LIN {X 0,Y 152.545,Z 875.411,A -85,B 0,C 180,E1 7963.211,E2 7963.211} C_VEL
LIN {X 0,Y 145.581,Z 982.767,A -85,B 0,C 180,E1 7954.617,E2 7954.617} C_VEL
LIN {X 0,Y 143.975,Z 1022.889,A -85,B 0,C 180,E1 7951.06,E2 7951.06} C_VEL
LIN {X 0,Y 142.78,Z 1041.292,A -85,B 0,C 180,E1 7948.656,E2 7948.656} C_VEL
LIN {X 0,Y 141.52,Z 1057.681,A -85,B 0,C 180,E1 7945.736,E2 7945.736} C_VEL
LIN {X 0,Y 140.296,Z 1073.463,A -85,B 0,C 180,E1 7942.12,E2 7942.12} C_VEL
LIN {X 0,Y 139.325,Z 1089.114,A -85,B 0,C 180,E1 7937.533,E2 7937.533} C_VEL
LIN {X 0,Y 138.945,Z 1102.914,A -85,B 0,C 180,E1 7932.458,E2 7932.458} C_VEL
LIN {X 0,Y 139.338,Z 1114.971,A -85,B 0,C 180,E1 7926.998,E2 7926.998} C_VEL
LIN {X 0,Y 141.002,Z 1126.172,A -85,B 0,C 180,E1 7920.804,E2 7920.804} C_VEL
LIN {X 0,Y 144.181,Z 1135.172,A -85,B 0,C 180,E1 7914.819,E2 7914.819} C_VEL
LIN {X 0,Y 149.717,Z 1143.18,A -85,B 0,C 180,E1 7908.434,E2 7908.434} C_VEL
LIN {X 0,Y 156.242,Z 1148.409,A -85,B 0,C 180,E1 7903.255,E2 7903.255} C_VEL
LIN {X 0,Y 163.588,Z 1152.185,A -85,B 0,C 180,E1 7898.854,E2 7898.854} C_VEL
LIN {X 0,Y 173.945,Z 1154.929,A -85,B 0,C 180,E1 7894.088,E2 7894.088} C_VEL
LIN {X 0,Y 185.649,Z 1155.901,A -85,B 0,C 180,E1 7889.934,E2 7889.934} C_VEL
LIN {X 0,Y 197.459,Z 1155.135,A -85,B 0,C 180,E1 7886.53,E2 7886.53} C_VEL
LIN {X 0,Y 181.8,Z 1159.577,A -85,B 0,C 180,E1 7882.364,E2 7882.364} C_VEL
LIN {X 0,Y 167.775,Z 1162.466,A -85,B 0,C 180,E1 7877.134,E2 7877.134} C_VEL
LIN {X 0,Y 156.152,Z 1163.814,A -85,B 0,C 180,E1 7870.771,E2 7870.771} C_VEL
LIN {X 0,Y 147.735,Z 1163.571,A -85,B 0,C 180,E1 7863.703,E2 7863.703} C_VEL
LIN {X 0,Y 142.553,Z 1161.973,A -85,B 0,C 180,E1 7855.771,E2 7855.771} C_VEL
LIN {X 0,Y 141.021,Z 1159.791,A -85,B 0,C 180,E1 7849.675,E2 7849.675} C_VEL
LIN {X 0,Y 139.075,Z 1166.656,A -85,B 0,C 180,E1 7844.994,E2 7844.994} C_VEL
LIN {X 0,Y 138.656,Z 1175.79,A -85,B 0,C 180,E1 7837.869,E2 7837.869} C_VEL
LIN {X 0,Y 139.015,Z 1182.334,A -85,B 0,C 180,E1 7831.643,E2 7831.643} C_VEL
LIN {X 0,Y 138.861,Z 1186.047,A -85,B 0,C 180,E1 7827.105,E2 7827.105} C_VEL
LIN {X 0,Y 138.143,Z 1190.598,A -85,B 0,C 180,E1 7819.569,E2 7819.569} C_VEL
LIN {X 0,Y 139.172,Z 1194.136,A -85,B 0,C 180,E1 7811.411,E2 7811.411} C_VEL
LIN {X 0,Y 139.307,Z 1194.975,A -85,B 0,C 180,E1 7808.234,E2 7808.234} C_VEL
LIN {X 0,Y 138.381,Z 1195.914,A -85,B 0,C 180,E1 7799.239,E2 7799.239} C_VEL
LIN {X 0,Y 139.856,Z 1196.329,A -85,B 0,C 180,E1 7796.802,E2 7796.802} C_VEL
LIN {X 0,Y 154.114,Z 1198.205,A -85,B 0,C 180,E1 7786.029,E2 7786.029} C_VEL
LIN {X 0,Y 160.613,Z 1198.418,A -85,B 0,C 180,E1 7782.633,E2 7782.633} C_VEL
LIN {X 0,Y 145.334,Z 1193.936,A -85,B 0,C 180,E1 7773.404,E2 7773.404} C_VEL
LIN {X 0,Y 135.187,Z 1187.729,A -85,B 0,C 180,E1 7762.629,E2 7762.629} C_VEL
LIN {X 0,Y 130.339,Z 1180.191,A -85,B 0,C 180,E1 7751.515,E2 7751.515} C_VEL
LIN {X 0,Y 129.225,Z 1173.64,A -85,B 0,C 180,E1 7743.558,E2 7743.558} C_VEL
LIN {X 0,Y 129.001,Z 1167.014,A -85,B 0,C 180,E1 7736.84,E2 7736.84} C_VEL
LIN {X 0,Y 129.423,Z 1158.193,A -85,B 0,C 180,E1 7729.324,E2 7729.324} C_VEL
LIN {X 0,Y 131.101,Z 1147.526,A -85,B 0,C 180,E1 7721.788,E2 7721.788} C_VEL
LIN {X 0,Y 134.817,Z 1133.432,A -85,B 0,C 180,E1 7713.588,E2 7713.588} C_VEL
LIN {X 0,Y 139.89,Z 1118.577,A -85,B 0,C 180,E1 7706.619,E2 7706.619} C_VEL
LIN {X 0,Y 146.552,Z 1101.226,A -85,B 0,C 180,E1 7700.12,E2 7700.12} C_VEL
LIN {X 0,Y 154.181,Z 1082.006,A -85,B 0,C 180,E1 7694.503,E2 7694.503} C_VEL
LIN {X 0,Y 162.11,Z 1061.669,A -85,B 0,C 180,E1 7689.847,E2 7689.847} C_VEL
LIN {X 0,Y 169.639,Z 1041.208,A -85,B 0,C 180,E1 7686.161,E2 7686.161} C_VEL
LIN {X 0,Y 177.085,Z 1019.188,A -85,B 0,C 180,E1 7683.034,E2 7683.034} C_VEL
LIN {X 0,Y 184.27,Z 995.291,A -85,B 0,C 180,E1 7680.387,E2 7680.387} C_VEL
LIN {X 0,Y 190.704,Z 970.389,A -85,B 0,C 180,E1 7678.271,E2 7678.271} C_VEL
LIN {X 0,Y 196.151,Z 944.496,A -85,B 0,C 180,E1 7676.635,E2 7676.635} C_VEL
LIN {X 0,Y 218.47,Z 820.524,A -85,B 0,C 180,E1 7670.985,E2 7670.985} C_VEL
LIN {X 0,Y 208.205,Z 799.294,A -85,B 0,C 180,E1 7666.295,E2 7666.295} C_VEL
LIN {X 0,Y 199.26,Z 781.915,A -85,B 0,C 180,E1 7661.693,E2 7661.693} C_VEL
LIN {X 0,Y 190.636,Z 766.045,A -85,B 0,C 180,E1 7656.63,E2 7656.63} C_VEL
LIN {X 0,Y 183.761,Z 754.052,A -85,B 0,C 180,E1 7652.031,E2 7652.031} C_VEL
LIN {X 0,Y 176.635,Z 742.307,A -85,B 0,C 180,E1 7646.516,E2 7646.516} C_VEL
LIN {X 0,Y 170.396,Z 732.497,A -85,B 0,C 180,E1 7640.701,E2 7640.701} C_VEL
LIN {X 0,Y 167.6,Z 728.346,A -85,B 0,C 180,E1 7637.728,E2 7637.728} C_VEL
LIN {X 0,Y 162.392,Z 733.212,A -85,B 0,C 180,E1 7634.397,E2 7634.397} C_VEL
LIN {X 0,Y 159.719,Z 736.002,A -85,B 0,C 180,E1 7632.518,E2 7632.518} C_VEL
LIN {X 0,Y 158.824,Z 736.981,A -85,B 0,C 180,E1 7631.893,E2 7631.893} C_VEL
LIN {X 0,Y 156.607,Z 739.804,A -85,B 0,C 180,E1 7630.324,E2 7630.324} C_VEL
LIN {X 0,Y 155.514,Z 740.538,A -85,B 0,C 180,E1 7629.198,E2 7629.198} C_VEL
LIN {X 0,Y 160.894,Z 759.966,A -85,B 0,C 180,E1 7624.021,E2 7624.021} C_VEL
LIN {X 0,Y 163.391,Z 771.027,A -85,B 0,C 180,E1 7621.395,E2 7621.395} C_VEL
LIN {X 0,Y 155.237,Z 815.549,A -85,B 0,C 180,E1 7614.124,E2 7614.124} C_VEL
LIN {X 0,Y 149.141,Z 851.757,A -85,B 0,C 180,E1 7607.907,E2 7607.907} C_VEL
LIN {X 0,Y 144.614,Z 876.252,A -85,B 0,C 180,E1 7603.729,E2 7603.729} C_VEL
LIN {X 0,Y 137.618,Z 981.604,A -85,B 0,C 180,E1 7594.762,E2 7594.762} C_VEL
LIN {X 0,Y 135.971,Z 1022.857,A -85,B 0,C 180,E1 7590.869,E2 7590.869} C_VEL
LIN {X 0,Y 134.825,Z 1040.561,A -85,B 0,C 180,E1 7588.477,E2 7588.477} C_VEL
LIN {X 0,Y 133.59,Z 1056.825,A -85,B 0,C 180,E1 7585.48,E2 7585.48} C_VEL
LIN {X 0,Y 132.34,Z 1073.426,A -85,B 0,C 180,E1 7581.486,E2 7581.486} C_VEL
LIN {X 0,Y 131.46,Z 1088.714,A -85,B 0,C 180,E1 7576.79,E2 7576.79} C_VEL
LIN {X 0,Y 131.178,Z 1102.082,A -85,B 0,C 180,E1 7571.663,E2 7571.663} C_VEL
LIN {X 0,Y 131.686,Z 1114.224,A -85,B 0,C 180,E1 7565.979,E2 7565.979} C_VEL
LIN {X 0,Y 133.357,Z 1124.834,A -85,B 0,C 180,E1 7559.991,E2 7559.991} C_VEL
LIN {X 0,Y 137.012,Z 1134.809,A -85,B 0,C 180,E1 7553.286,E2 7553.286} C_VEL
LIN {X 0,Y 142.58,Z 1142.712,A -85,B 0,C 180,E1 7547.023,E2 7547.023} C_VEL
LIN {X 0,Y 149.715,Z 1148.569,A -85,B 0,C 180,E1 7541.488,E2 7541.488} C_VEL
LIN {X 0,Y 158.954,Z 1153.231,A -85,B 0,C 180,E1 7536.252,E2 7536.252} C_VEL
LIN {X 0,Y 170.023,Z 1156.128,A -85,B 0,C 180,E1 7531.545,E2 7531.545} C_VEL
LIN {X 0,Y 182.808,Z 1157.266,A -85,B 0,C 180,E1 7527.377,E2 7527.377} C_VEL
LIN {X 0,Y 185.108,Z 1157.286,A -85,B 0,C 180,E1 7526.647,E2 7526.647} C_VEL
LIN {X 0,Y 169.803,Z 1160.339,A -85,B 0,C 180,E1 7522.089,E2 7522.089} C_VEL
LIN {X 0,Y 155.982,Z 1161.959,A -85,B 0,C 180,E1 7516.177,E2 7516.177} C_VEL
LIN {X 0,Y 145.322,Z 1162.022,A -85,B 0,C 180,E1 7509.265,E2 7509.265} C_VEL
LIN {X 0,Y 137.39,Z 1160.473,A -85,B 0,C 180,E1 7500.62,E2 7500.62} C_VEL
LIN {X 0,Y 133.942,Z 1157.464,A -85,B 0,C 180,E1 7491.91,E2 7491.91} C_VEL
LIN {X 0,Y 133.735,Z 1156.95,A -85,B 0,C 180,E1 7490.567,E2 7490.567} C_VEL
LIN {X 0,Y 131.347,Z 1164.22,A -85,B 0,C 180,E1 7485.446,E2 7485.446} C_VEL
LIN {X 0,Y 130.903,Z 1173.526,A -85,B 0,C 180,E1 7477.897,E2 7477.897} C_VEL
LIN {X 0,Y 131.3,Z 1179.858,A -85,B 0,C 180,E1 7471.74,E2 7471.74} C_VEL
LIN {X 0,Y 131.259,Z 1183.443,A -85,B 0,C 180,E1 7467.374,E2 7467.374} C_VEL
LIN {X 0,Y 130.553,Z 1187.547,A -85,B 0,C 180,E1 7460.739,E2 7460.739} C_VEL
LIN {X 0,Y 131.554,Z 1192.034,A -85,B 0,C 180,E1 7450.888,E2 7450.888} C_VEL
LIN {X 0,Y 138.235,Z 1195.9,A -85,B 0,C 180,E1 7438.608,E2 7438.608} C_VEL
LIN {X 0,Y 139.856,Z 1196.329,A -85,B 0,C 180,E1 7436.802,E2 7436.802} C_VEL
LIN {X 0,Y 141.939,Z 1196.799,A -85,B 0,C 180,E1 7433.764,E2 7433.764} C_VEL
LIN {X 0,Y 146.454,Z 1196.812,A -85,B 0,C 180,E1 7425.511,E2 7425.511} C_VEL
LIN {X 0,Y 149.63,Z 1196.99,A -85,B 0,C 180,E1 7423.251,E2 7423.251} C_VEL
LIN {X 0,Y 150.631,Z 1197.048,A -85,B 0,C 180,E1 7422.626,E2 7422.626} C_VEL
LIN {X 0,Y 135.976,Z 1191.87,A -85,B 0,C 180,E1 7412.977,E2 7412.977} C_VEL
LIN {X 0,Y 126.267,Z 1184.926,A -85,B 0,C 180,E1 7401.372,E2 7401.372} C_VEL
LIN {X 0,Y 122.321,Z 1177.694,A -85,B 0,C 180,E1 7390.847,E2 7390.847} C_VEL
LIN {X 0,Y 121.327,Z 1170.66,A -85,B 0,C 180,E1 7382.372,E2 7382.372} C_VEL
LIN {X 0,Y 121.176,Z 1163.572,A -85,B 0,C 180,E1 7375.277,E2 7375.277} C_VEL
LIN {X 0,Y 121.794,Z 1154.615,A -85,B 0,C 180,E1 7367.686,E2 7367.686} C_VEL
LIN {X 0,Y 124.035,Z 1142.661,A -85,B 0,C 180,E1 7359.236,E2 7359.236} C_VEL
LIN {X 0,Y 127.925,Z 1129.407,A -85,B 0,C 180,E1 7351.536,E2 7351.536} C_VEL
LIN {X 0,Y 133.683,Z 1113.533,A -85,B 0,C 180,E1 7344.169,E2 7344.169} C_VEL
LIN {X 0,Y 140.64,Z 1096.154,A -85,B 0,C 180,E1 7337.803,E2 7337.803} C_VEL
LIN {X 0,Y 148.56,Z 1076.816,A -85,B 0,C 180,E1 7332.252,E2 7332.252} C_VEL
LIN {X 0,Y 156.67,Z 1056.425,A -85,B 0,C 180,E1 7327.699,E2 7327.699} C_VEL
LIN {X 0,Y 164.608,Z 1035.106,A -85,B 0,C 180,E1 7323.981,E2 7323.981} C_VEL
LIN {X 0,Y 172.371,Z 1012.171,A -85,B 0,C 180,E1 7320.865,E2 7320.865} C_VEL
LIN {X 0,Y 179.199,Z 989.294,A -85,B 0,C 180,E1 7318.458,E2 7318.458} C_VEL
LIN {X 0,Y 185.667,Z 963.62,A -85,B 0,C 180,E1 7316.403,E2 7316.403} C_VEL
LIN {X 0,Y 191.114,Z 937.113,A -85,B 0,C 180,E1 7314.846,E2 7314.846} C_VEL
LIN {X 0,Y 212.132,Z 823.264,A -85,B 0,C 180,E1 7309.63,E2 7309.63} C_VEL
LIN {X 0,Y 202.61,Z 803.298,A -85,B 0,C 180,E1 7305.02,E2 7305.02} C_VEL
LIN {X 0,Y 194.23,Z 786.71,A -85,B 0,C 180,E1 7300.452,E2 7300.452} C_VEL
LIN {X 0,Y 186.023,Z 771.345,A -85,B 0,C 180,E1 7295.402,E2 7295.402} C_VEL
LIN {X 0,Y 179.795,Z 760.212,A -85,B 0,C 180,E1 7291.009,E2 7291.009} C_VEL
LIN {X 0,Y 173.113,Z 748.879,A -85,B 0,C 180,E1 7285.532,E2 7285.532} C_VEL
LIN {X 0,Y 167.239,Z 739.438,A -85,B 0,C 180,E1 7279.846,E2 7279.846} C_VEL
LIN {X 0,Y 165.416,Z 737.027,A -85,B 0,C 180,E1 7277.905,E2 7277.905} C_VEL
LIN {X 0,Y 161.748,Z 740.522,A -85,B 0,C 180,E1 7275.639,E2 7275.639} C_VEL
LIN {X 0,Y 158.335,Z 744.095,A -85,B 0,C 180,E1 7273.334,E2 7273.334} C_VEL
LIN {X 0,Y 155.532,Z 747.222,A -85,B 0,C 180,E1 7271.362,E2 7271.362} C_VEL
LIN {X 0,Y 154.661,Z 748.187,A -85,B 0,C 180,E1 7270.689,E2 7270.689} C_VEL
LIN {X 0,Y 152.41,Z 751.457,A -85,B 0,C 180,E1 7269.056,E2 7269.056} C_VEL
LIN {X 0,Y 151.088,Z 752.484,A -85,B 0,C 180,E1 7267.696,E2 7267.696} C_VEL
LIN {X 0,Y 155.914,Z 771.479,A -85,B 0,C 180,E1 7262.714,E2 7262.714} C_VEL
LIN {X 0,Y 155.794,Z 773.532,A -85,B 0,C 180,E1 7262.317,E2 7262.317} C_VEL
LIN {X 0,Y 147.3,Z 818.296,A -85,B 0,C 180,E1 7254.768,E2 7254.768} C_VEL
LIN {X 0,Y 141.451,Z 851.732,A -85,B 0,C 180,E1 7248.821,E2 7248.821} C_VEL
LIN {X 0,Y 136.669,Z 877.206,A -85,B 0,C 180,E1 7244.271,E2 7244.271} C_VEL
LIN {X 0,Y 129.58,Z 982.567,A -85,B 0,C 180,E1 7234.691,E2 7234.691} C_VEL
LIN {X 0,Y 127.954,Z 1023.158,A -85,B 0,C 180,E1 7230.581,E2 7230.581} C_VEL
LIN {X 0,Y 126.826,Z 1040.595,A -85,B 0,C 180,E1 7228.086,E2 7228.086} C_VEL
LIN {X 0,Y 125.565,Z 1057.39,A -85,B 0,C 180,E1 7224.815,E2 7224.815} C_VEL
LIN {X 0,Y 124.407,Z 1073.471,A -85,B 0,C 180,E1 7220.699,E2 7220.699} C_VEL
LIN {X 0,Y 123.634,Z 1088.566,A -85,B 0,C 180,E1 7215.786,E2 7215.786} C_VEL
LIN {X 0,Y 123.468,Z 1101.769,A -85,B 0,C 180,E1 7210.488,E2 7210.488} C_VEL
LIN {X 0,Y 124.25,Z 1114.595,A -85,B 0,C 180,E1 7204.143,E2 7204.143} C_VEL
LIN {X 0,Y 126.348,Z 1125.444,A -85,B 0,C 180,E1 7197.723,E2 7197.723} C_VEL
LIN {X 0,Y 130.727,Z 1135.641,A -85,B 0,C 180,E1 7190.595,E2 7190.595} C_VEL
LIN {X 0,Y 136.868,Z 1143.476,A -85,B 0,C 180,E1 7184.309,E2 7184.309} C_VEL
LIN {X 0,Y 145.074,Z 1149.665,A -85,B 0,C 180,E1 7178.489,E2 7178.489} C_VEL
LIN {X 0,Y 155.333,Z 1154.452,A -85,B 0,C 180,E1 7173.21,E2 7173.21} C_VEL
LIN {X 0,Y 167.2,Z 1157.426,A -85,B 0,C 180,E1 7168.641,E2 7168.641} C_VEL
LIN {X 0,Y 172.939,Z 1158.217,A -85,B 0,C 180,E1 7166.739,E2 7166.739} C_VEL
LIN {X 0,Y 157.28,Z 1160.043,A -85,B 0,C 180,E1 7161.431,E2 7161.431} C_VEL
LIN {X 0,Y 144.409,Z 1160.358,A -85,B 0,C 180,E1 7154.922,E2 7154.922} C_VEL
LIN {X 0,Y 133.323,Z 1158.865,A -85,B 0,C 180,E1 7145.794,E2 7145.794} C_VEL
LIN {X 0,Y 127.765,Z 1155.911,A -85,B 0,C 180,E1 7136.485,E2 7136.485} C_VEL
LIN {X 0,Y 126.566,Z 1153.907,A -85,B 0,C 180,E1 7131.546,E2 7131.546} C_VEL
LIN {X 0,Y 123.81,Z 1160.941,A -85,B 0,C 180,E1 7126.412,E2 7126.412} C_VEL
LIN {X 0,Y 123.155,Z 1171.322,A -85,B 0,C 180,E1 7117.834,E2 7117.834} C_VEL
LIN {X 0,Y 123.626,Z 1177.712,A -85,B 0,C 180,E1 7111.384,E2 7111.384} C_VEL
LIN {X 0,Y 123.613,Z 1181.117,A -85,B 0,C 180,E1 7107.212,E2 7107.212} C_VEL
LIN {X 0,Y 122.888,Z 1185.844,A -85,B 0,C 180,E1 7099.208,E2 7099.208} C_VEL
LIN {X 0,Y 124.776,Z 1190.699,A -85,B 0,C 180,E1 7087.868,E2 7087.868} C_VEL
LIN {X 0,Y 132.666,Z 1194.586,A -85,B 0,C 180,E1 7075.522,E2 7075.522} C_VEL
LIN {X 0,Y 146.701,Z 1196.742,A -85,B 0,C 180,E1 7064.852,E2 7064.852} C_VEL
LIN {X 0,Y 149.63,Z 1196.99,A -85,B 0,C 180,E1 7063.251,E2 7063.251} C_VEL
LIN {X 0,Y 149.771,Z 1196.868,A -85,B 0,C 180,E1 7062.441,E2 7062.441} C_VEL
LIN {X 0,Y 148.075,Z 1196.388,A -85,B 0,C 180,E1 7061.462,E2 7061.462} C_VEL
LIN {X 0,Y 144.076,Z 1195.428,A -85,B 0,C 180,E1 7060.353,E2 7060.353} C_VEL
LIN {X 0,Y 134.991,Z 1193.082,A -85,B 0,C 180,E1 7058.39,E2 7058.39} C_VEL
LIN {X 0,Y 131.931,Z 1192.058,A -85,B 0,C 180,E1 7056.952,E2 7056.952} C_VEL
LIN {X 0,Y 120.505,Z 1185.095,A -85,B 0,C 180,E1 7045.241,E2 7045.241} C_VEL
LIN {X 0,Y 114.994,Z 1177.091,A -85,B 0,C 180,E1 7033.077,E2 7033.077} C_VEL
LIN {X 0,Y 113.65,Z 1170.011,A -85,B 0,C 180,E1 7024.047,E2 7024.047} C_VEL
LIN {X 0,Y 113.353,Z 1163.295,A -85,B 0,C 180,E1 7016.839,E2 7016.839} C_VEL
LIN {X 0,Y 113.765,Z 1154.541,A -85,B 0,C 180,E1 7008.862,E2 7008.862} C_VEL
LIN {X 0,Y 115.856,Z 1142.609,A -85,B 0,C 180,E1 6999.817,E2 6999.817} C_VEL
LIN {X 0,Y 119.724,Z 1129.381,A -85,B 0,C 180,E1 6991.585,E2 6991.585} C_VEL
LIN {X 0,Y 125.476,Z 1113.805,A -85,B 0,C 180,E1 6983.878,E2 6983.878} C_VEL
LIN {X 0,Y 132.489,Z 1096.741,A -85,B 0,C 180,E1 6977.231,E2 6977.231} C_VEL
LIN {X 0,Y 140.602,Z 1077.546,A -85,B 0,C 180,E1 6971.411,E2 6971.411} C_VEL
LIN {X 0,Y 149.251,Z 1056.491,A -85,B 0,C 180,E1 6966.509,E2 6966.509} C_VEL
LIN {X 0,Y 157.734,Z 1034.393,A -85,B 0,C 180,E1 6962.548,E2 6962.548} C_VEL
LIN {X 0,Y 165.401,Z 1012.337,A -85,B 0,C 180,E1 6959.499,E2 6959.499} C_VEL
LIN {X 0,Y 172.718,Z 988.427,A -85,B 0,C 180,E1 6956.953,E2 6956.953} C_VEL
LIN {X 0,Y 179.231,Z 963.253,A -85,B 0,C 180,E1 6954.915,E2 6954.915} C_VEL
LIN {X 0,Y 184.757,Z 937.115,A -85,B 0,C 180,E1 6953.361,E2 6953.361} C_VEL
LIN {X 0,Y 205.928,Z 826.034,A -85,B 0,C 180,E1 6948.209,E2 6948.209} C_VEL
LIN {X 0,Y 196.018,Z 805.096,A -85,B 0,C 180,E1 6943.124,E2 6943.124} C_VEL
LIN {X 0,Y 187.656,Z 788.383,A -85,B 0,C 180,E1 6938.199,E2 6938.199} C_VEL
LIN {X 0,Y 179.817,Z 773.471,A -85,B 0,C 180,E1 6932.913,E2 6932.913} C_VEL
LIN {X 0,Y 173.81,Z 762.774,A -85,B 0,C 180,E1 6928.274,E2 6928.274} C_VEL
LIN {X 0,Y 168.474,Z 753.77,A -85,B 0,C 180,E1 6923.53,E2 6923.53} C_VEL
LIN {X 0,Y 164.045,Z 746.262,A -85,B 0,C 180,E1 6918.865,E2 6918.865} C_VEL
LIN {X 0,Y 163.406,Z 745.624,A -85,B 0,C 180,E1 6918.208,E2 6918.208} C_VEL
LIN {X 0,Y 157.789,Z 751.248,A -85,B 0,C 180,E1 6914.717,E2 6914.717} C_VEL
LIN {X 0,Y 154.217,Z 755.191,A -85,B 0,C 180,E1 6912.264,E2 6912.264} C_VEL
LIN {X 0,Y 151.528,Z 758.646,A -85,B 0,C 180,E1 6910.34,E2 6910.34} C_VEL
LIN {X 0,Y 150.314,Z 760.001,A -85,B 0,C 180,E1 6909.312,E2 6909.312} C_VEL
LIN {X 0,Y 147.907,Z 763.623,A -85,B 0,C 180,E1 6907.563,E2 6907.563} C_VEL
LIN {X 0,Y 146.552,Z 764.968,A -85,B 0,C 180,E1 6906.034,E2 6906.034} C_VEL
LIN {X 0,Y 148.624,Z 774.15,A -85,B 0,C 180,E1 6903.645,E2 6903.645} C_VEL
LIN {X 0,Y 139.904,Z 818.134,A -85,B 0,C 180,E1 6895.984,E2 6895.984} C_VEL
LIN {X 0,Y 133.933,Z 850.931,A -85,B 0,C 180,E1 6889.911,E2 6889.911} C_VEL
LIN {X 0,Y 128.735,Z 877.891,A -85,B 0,C 180,E1 6884.844,E2 6884.844} C_VEL
LIN {X 0,Y 121.611,Z 981.542,A -85,B 0,C 180,E1 6874.745,E2 6874.745} C_VEL
LIN {X 0,Y 119.971,Z 1022.989,A -85,B 0,C 180,E1 6870.273,E2 6870.273} C_VEL
LIN {X 0,Y 118.863,Z 1040.253,A -85,B 0,C 180,E1 6867.683,E2 6867.683} C_VEL
LIN {X 0,Y 117.593,Z 1057.641,A -85,B 0,C 180,E1 6864.076,E2 6864.076} C_VEL
LIN {X 0,Y 116.474,Z 1074.17,A -85,B 0,C 180,E1 6859.549,E2 6859.549} C_VEL
LIN {X 0,Y 115.87,Z 1088.027,A -85,B 0,C 180,E1 6854.762,E2 6854.762} C_VEL
LIN {X 0,Y 115.878,Z 1102.165,A -85,B 0,C 180,E1 6848.728,E2 6848.728} C_VEL
LIN {X 0,Y 116.867,Z 1114.218,A -85,B 0,C 180,E1 6842.441,E2 6842.441} C_VEL
LIN {X 0,Y 119.569,Z 1125.934,A -85,B 0,C 180,E1 6835.193,E2 6835.193} C_VEL
LIN {X 0,Y 124.506,Z 1136.018,A -85,B 0,C 180,E1 6827.938,E2 6827.938} C_VEL
LIN {X 0,Y 132.005,Z 1144.596,A -85,B 0,C 180,E1 6820.982,E2 6820.982} C_VEL
LIN {X 0,Y 141.584,Z 1151.073,A -85,B 0,C 180,E1 6814.921,E2 6814.921} C_VEL
LIN {X 0,Y 152.901,Z 1155.882,A -85,B 0,C 180,E1 6809.757,E2 6809.757} C_VEL
LIN {X 0,Y 160.969,Z 1158.005,A -85,B 0,C 180,E1 6806.78,E2 6806.78} C_VEL
LIN {X 0,Y 145.565,Z 1158.571,A -85,B 0,C 180,E1 6800.796,E2 6800.796} C_VEL
LIN {X 0,Y 130.941,Z 1157.271,A -85,B 0,C 180,E1 6791.54,E2 6791.54} C_VEL
LIN {X 0,Y 122.799,Z 1154.407,A -85,B 0,C 180,E1 6781.948,E2 6781.948} C_VEL
LIN {X 0,Y 119.571,Z 1150.659,A -85,B 0,C 180,E1 6772.745,E2 6772.745} C_VEL
LIN {X 0,Y 116.216,Z 1158.257,A -85,B 0,C 180,E1 6767.002,E2 6767.002} C_VEL
LIN {X 0,Y 115.44,Z 1169.328,A -85,B 0,C 180,E1 6757.458,E2 6757.458} C_VEL
LIN {X 0,Y 116.017,Z 1175.925,A -85,B 0,C 180,E1 6750.487,E2 6750.487} C_VEL
LIN {X 0,Y 115.924,Z 1179.23,A -85,B 0,C 180,E1 6746.037,E2 6746.037} C_VEL
LIN {X 0,Y 115.348,Z 1184.244,A -85,B 0,C 180,E1 6736.968,E2 6736.968} C_VEL
LIN {X 0,Y 118.617,Z 1189.473,A -85,B 0,C 180,E1 6723.995,E2 6723.995} C_VEL
LIN {X 0,Y 127.906,Z 1193.185,A -85,B 0,C 180,E1 6711.854,E2 6711.854} C_VEL
LIN {X 0,Y 140.818,Z 1195.288,A -85,B 0,C 180,E1 6702.671,E2 6702.671} C_VEL
LIN {X 0,Y 131.931,Z 1192.058,A -85,B 0,C 180,E1 6696.952,E2 6696.952} C_VEL
LIN {X 0,Y 127.499,Z 1190.265,A -85,B 0,C 180,E1 6694.249,E2 6694.249} C_VEL
LIN {X 0,Y 114.215,Z 1183.944,A -85,B 0,C 180,E1 6686.961,E2 6686.961} C_VEL
LIN {X 0,Y 111.564,Z 1181.851,A -85,B 0,C 180,E1 6684.039,E2 6684.039} C_VEL
LIN {X 0,Y 107.035,Z 1174.16,A -85,B 0,C 180,E1 6672.419,E2 6672.419} C_VEL
LIN {X 0,Y 105.781,Z 1166.674,A -85,B 0,C 180,E1 6662.721,E2 6662.721} C_VEL
LIN {X 0,Y 105.559,Z 1159.013,A -85,B 0,C 180,E1 6654.577,E2 6654.577} C_VEL
LIN {X 0,Y 106.381,Z 1149.317,A -85,B 0,C 180,E1 6645.867,E2 6645.867} C_VEL
LIN {X 0,Y 109.024,Z 1137.287,A -85,B 0,C 180,E1 6636.787,E2 6636.787} C_VEL
LIN {X 0,Y 113.713,Z 1123.117,A -85,B 0,C 180,E1 6628.171,E2 6628.171} C_VEL
LIN {X 0,Y 120.362,Z 1106.532,A -85,B 0,C 180,E1 6620.248,E2 6620.248} C_VEL
LIN {X 0,Y 128.242,Z 1088.34,A -85,B 0,C 180,E1 6613.537,E2 6613.537} C_VEL
LIN {X 0,Y 136.875,Z 1068.437,A -85,B 0,C 180,E1 6607.928,E2 6607.928} C_VEL
LIN {X 0,Y 145.527,Z 1047.57,A -85,B 0,C 180,E1 6603.422,E2 6603.422} C_VEL
LIN {X 0,Y 153.942,Z 1025.464,A -85,B 0,C 180,E1 6599.769,E2 6599.769} C_VEL
LIN {X 0,Y 161.999,Z 1001.826,A -85,B 0,C 180,E1 6596.785,E2 6596.785} C_VEL
LIN {X 0,Y 169.185,Z 977.425,A -85,B 0,C 180,E1 6594.442,E2 6594.442} C_VEL
LIN {X 0,Y 175.516,Z 951.425,A -85,B 0,C 180,E1 6592.598,E2 6592.598} C_VEL
LIN {X 0,Y 199.679,Z 828.821,A -85,B 0,C 180,E1 6586.722,E2 6586.722} C_VEL
LIN {X 0,Y 190.422,Z 808.771,A -85,B 0,C 180,E1 6581.629,E2 6581.629} C_VEL
LIN {X 0,Y 181.964,Z 791.617,A -85,B 0,C 180,E1 6576.314,E2 6576.314} C_VEL
LIN {X 0,Y 174.769,Z 777.605,A -85,B 0,C 180,E1 6571.07,E2 6571.07} C_VEL
LIN {X 0,Y 168.373,Z 765.961,A -85,B 0,C 180,E1 6565.654,E2 6565.654} C_VEL
LIN {X 0,Y 162.703,Z 756.306,A -85,B 0,C 180,E1 6559.998,E2 6559.998} C_VEL
LIN {X 0,Y 161.468,Z 754.227,A -85,B 0,C 180,E1 6558.576,E2 6558.576} C_VEL
LIN {X 0,Y 157.097,Z 758.635,A -85,B 0,C 180,E1 6555.953,E2 6555.953} C_VEL
LIN {X 0,Y 153.81,Z 762.248,A -85,B 0,C 180,E1 6553.773,E2 6553.773} C_VEL
LIN {X 0,Y 150.588,Z 765.962,A -85,B 0,C 180,E1 6551.531,E2 6551.531} C_VEL
LIN {X 0,Y 147.001,Z 770.844,A -85,B 0,C 180,E1 6548.875,E2 6548.875} C_VEL
LIN {X 0,Y 145.762,Z 772.27,A -85,B 0,C 180,E1 6547.804,E2 6547.804} C_VEL
LIN {X 0,Y 143.37,Z 776.355,A -85,B 0,C 180,E1 6545.986,E2 6545.986} C_VEL
LIN {X 0,Y 142.023,Z 779.335,A -85,B 0,C 180,E1 6545.118,E2 6545.118} C_VEL
LIN {X 0,Y 139.02,Z 786.157,A -85,B 0,C 180,E1 6543.063,E2 6543.063} C_VEL
LIN {X 0,Y 130.105,Z 830.483,A -85,B 0,C 180,E1 6534.914,E2 6534.914} C_VEL
LIN {X 0,Y 126.204,Z 851.091,A -85,B 0,C 180,E1 6530.918,E2 6530.918} C_VEL
LIN {X 0,Y 120.796,Z 878.663,A -85,B 0,C 180,E1 6525.456,E2 6525.456} C_VEL
LIN {X 0,Y 113.618,Z 981.222,A -85,B 0,C 180,E1 6514.71,E2 6514.71} C_VEL
LIN {X 0,Y 112.017,Z 1022.578,A -85,B 0,C 180,E1 6509.885,E2 6509.885} C_VEL
LIN {X 0,Y 110.892,Z 1040.325,A -85,B 0,C 180,E1 6507.074,E2 6507.074} C_VEL
LIN {X 0,Y 109.62,Z 1058.308,A -85,B 0,C 180,E1 6503.08,E2 6503.08} C_VEL
LIN {X 0,Y 108.617,Z 1074.672,A -85,B 0,C 180,E1 6498.227,E2 6498.227} C_VEL
LIN {X 0,Y 108.152,Z 1089.225,A -85,B 0,C 180,E1 6492.808,E2 6492.808} C_VEL
LIN {X 0,Y 108.468,Z 1103.18,A -85,B 0,C 180,E1 6486.339,E2 6486.339} C_VEL
LIN {X 0,Y 109.934,Z 1115.448,A -85,B 0,C 180,E1 6479.468,E2 6479.468} C_VEL
LIN {X 0,Y 113.644,Z 1127.737,A -85,B 0,C 180,E1 6471.387,E2 6471.387} C_VEL
LIN {X 0,Y 120.044,Z 1138.176,A -85,B 0,C 180,E1 6463.538,E2 6463.538} C_VEL
LIN {X 0,Y 128.779,Z 1146.491,A -85,B 0,C 180,E1 6456.663,E2 6456.663} C_VEL
LIN {X 0,Y 138.824,Z 1152.478,A -85,B 0,C 180,E1 6451.137,E2 6451.137} C_VEL
LIN {X 0,Y 149.361,Z 1156.728,A -85,B 0,C 180,E1 6446.793,E2 6446.793} C_VEL
LIN {X 0,Y 133.713,Z 1156.014,A -85,B 0,C 180,E1 6439.697,E2 6439.697} C_VEL
LIN {X 0,Y 121.973,Z 1153.849,A -85,B 0,C 180,E1 6430.972,E2 6430.972} C_VEL
LIN {X 0,Y 114.814,Z 1150.184,A -85,B 0,C 180,E1 6420.91,E2 6420.91} C_VEL
LIN {X 0,Y 112.702,Z 1147.284,A -85,B 0,C 180,E1 6414.078,E2 6414.078} C_VEL
LIN {X 0,Y 108.882,Z 1154.803,A -85,B 0,C 180,E1 6408.186,E2 6408.186} C_VEL
LIN {X 0,Y 107.736,Z 1166.174,A -85,B 0,C 180,E1 6397.995,E2 6397.995} C_VEL
LIN {X 0,Y 108.372,Z 1173.118,A -85,B 0,C 180,E1 6390.521,E2 6390.521} C_VEL
LIN {X 0,Y 108.443,Z 1176.273,A -85,B 0,C 180,E1 6386.292,E2 6386.292} C_VEL
LIN {X 0,Y 107.827,Z 1181.02,A -85,B 0,C 180,E1 6377.678,E2 6377.678} C_VEL
LIN {X 0,Y 110.243,Z 1186.181,A -85,B 0,C 180,E1 6365.334,E2 6365.334} C_VEL
LIN {X 0,Y 119.911,Z 1190.807,A -85,B 0,C 180,E1 6351.281,E2 6351.281} C_VEL
LIN {X 0,Y 131.134,Z 1193.062,A -85,B 0,C 180,E1 6342.747,E2 6342.747} C_VEL
LIN {X 0,Y 116.603,Z 1186.077,A -85,B 0,C 180,E1 6330.976,E2 6330.976} C_VEL
LIN {X 0,Y 111.564,Z 1181.851,A -85,B 0,C 180,E1 6324.039,E2 6324.039} C_VEL
LIN {X 0,Y 108.776,Z 1179.344,A -85,B 0,C 180,E1 6320.53,E2 6320.53} C_VEL
LIN {X 0,Y 101.748,Z 1173.204,A -85,B 0,C 180,E1 6313.671,E2 6313.671} C_VEL
LIN {X 0,Y 98.734,Z 1168.898,A -85,B 0,C 180,E1 6308.707,E2 6308.707} C_VEL
LIN {X 0,Y 98.479,Z 1168.004,A -85,B 0,C 180,E1 6307.516,E2 6307.516} C_VEL
LIN {X 0,Y 97.836,Z 1160.903,A -85,B 0,C 180,E1 6298.841,E2 6298.841} C_VEL
LIN {X 0,Y 98.067,Z 1151.639,A -85,B 0,C 180,E1 6289.438,E2 6289.438} C_VEL
LIN {X 0,Y 99.893,Z 1140.77,A -85,B 0,C 180,E1 6280.117,E2 6280.117} C_VEL
LIN {X 0,Y 104.262,Z 1126.396,A -85,B 0,C 180,E1 6270.101,E2 6270.101} C_VEL
LIN {X 0,Y 110.599,Z 1110.476,A -85,B 0,C 180,E1 6261.421,E2 6261.421} C_VEL
LIN {X 0,Y 118.345,Z 1093.012,A -85,B 0,C 180,E1 6254.114,E2 6254.114} C_VEL
LIN {X 0,Y 127.575,Z 1072.554,A -85,B 0,C 180,E1 6247.682,E2 6247.682} C_VEL
LIN {X 0,Y 136.68,Z 1051.5,A -85,B 0,C 180,E1 6242.742,E2 6242.742} C_VEL
LIN {X 0,Y 145.523,Z 1029.38,A -85,B 0,C 180,E1 6238.809,E2 6238.809} C_VEL
LIN {X 0,Y 153.704,Z 1006.639,A -85,B 0,C 180,E1 6235.733,E2 6235.733} C_VEL
LIN {X 0,Y 161.299,Z 982.271,A -85,B 0,C 180,E1 6233.242,E2 6233.242} C_VEL
LIN {X 0,Y 167.858,Z 957.178,A -85,B 0,C 180,E1 6231.318,E2 6231.318} C_VEL
LIN {X 0,Y 175.818,Z 919.286,A -85,B 0,C 180,E1 6229.219,E2 6229.219} C_VEL
LIN {X 0,Y 193.548,Z 831.584,A -85,B 0,C 180,E1 6225.165,E2 6225.165} C_VEL
LIN {X 0,Y 184.774,Z 812.323,A -85,B 0,C 180,E1 6220.022,E2 6220.022} C_VEL
LIN {X 0,Y 176.793,Z 795.738,A -85,B 0,C 180,E1 6214.627,E2 6214.627} C_VEL
LIN {X 0,Y 170.22,Z 782.665,A -85,B 0,C 180,E1 6209.5,E2 6209.5} C_VEL
LIN {X 0,Y 164.707,Z 772.306,A -85,B 0,C 180,E1 6204.527,E2 6204.527} C_VEL
LIN {X 0,Y 159.468,Z 762.996,A -85,B 0,C 180,E1 6198.934,E2 6198.934} C_VEL
LIN {X 0,Y 153.537,Z 769.125,A -85,B 0,C 180,E1 6195.344,E2 6195.344} C_VEL
LIN {X 0,Y 149.43,Z 773.913,A -85,B 0,C 180,E1 6192.609,E2 6192.609} C_VEL
LIN {X 0,Y 146.216,Z 778.003,A -85,B 0,C 180,E1 6190.241,E2 6190.241} C_VEL
LIN {X 0,Y 145.087,Z 779.595,A -85,B 0,C 180,E1 6189.429,E2 6189.429} C_VEL
LIN {X 0,Y 142.943,Z 783.128,A -85,B 0,C 180,E1 6187.941,E2 6187.941} C_VEL
LIN {X 0,Y 139.255,Z 791.242,A -85,B 0,C 180,E1 6185.744,E2 6185.744} C_VEL
LIN {X 0,Y 128.983,Z 818.402,A -85,B 0,C 180,E1 6180.514,E2 6180.514} C_VEL
LIN {X 0,Y 122.726,Z 835.555,A -85,B 0,C 180,E1 6176.112,E2 6176.112} C_VEL
LIN {X 0,Y 120.446,Z 841.963,A -85,B 0,C 180,E1 6173.894,E2 6173.894} C_VEL
LIN {X 0,Y 117.7,Z 854.406,A -85,B 0,C 180,E1 6171.385,E2 6171.385} C_VEL
LIN {X 0,Y 112.771,Z 880.165,A -85,B 0,C 180,E1 6166.002,E2 6166.002} C_VEL
LIN {X 0,Y 105.608,Z 981.467,A -85,B 0,C 180,E1 6154.531,E2 6154.531} C_VEL
LIN {X 0,Y 104.056,Z 1022.541,A -85,B 0,C 180,E1 6149.352,E2 6149.352} C_VEL
LIN {X 0,Y 102.922,Z 1040.83,A -85,B 0,C 180,E1 6146.22,E2 6146.22} C_VEL
LIN {X 0,Y 101.723,Z 1058.684,A -85,B 0,C 180,E1 6141.919,E2 6141.919} C_VEL
LIN {X 0,Y 100.87,Z 1074.251,A -85,B 0,C 180,E1 6136.99,E2 6136.99} C_VEL
LIN {X 0,Y 100.581,Z 1089.518,A -85,B 0,C 180,E1 6130.875,E2 6130.875} C_VEL
LIN {X 0,Y 101.202,Z 1103.427,A -85,B 0,C 180,E1 6123.953,E2 6123.953} C_VEL
LIN {X 0,Y 103.164,Z 1115.914,A -85,B 0,C 180,E1 6116.516,E2 6116.516} C_VEL
LIN {X 0,Y 107.559,Z 1127.987,A -85,B 0,C 180,E1 6108.187,E2 6108.187} C_VEL
LIN {X 0,Y 114.335,Z 1137.991,A -85,B 0,C 180,E1 6100.579,E2 6100.579} C_VEL
LIN {X 0,Y 123.955,Z 1146.672,A -85,B 0,C 180,E1 6093.542,E2 6093.542} C_VEL
LIN {X 0,Y 135.266,Z 1153.228,A -85,B 0,C 180,E1 6087.834,E2 6087.834} C_VEL
LIN {X 0,Y 137.921,Z 1154.377,A -85,B 0,C 180,E1 6086.659,E2 6086.659} C_VEL
LIN {X 0,Y 125.063,Z 1153.011,A -85,B 0,C 180,E1 6080.121,E2 6080.121} C_VEL
LIN {X 0,Y 113.621,Z 1149.882,A -85,B 0,C 180,E1 6070.624,E2 6070.624} C_VEL
LIN {X 0,Y 106.98,Z 1145.145,A -85,B 0,C 180,E1 6059.07,E2 6059.07} C_VEL
LIN {X 0,Y 106.117,Z 1143.584,A -85,B 0,C 180,E1 6055.677,E2 6055.677} C_VEL
LIN {X 0,Y 101.944,Z 1150.566,A -85,B 0,C 180,E1 6050.069,E2 6050.069} C_VEL
LIN {X 0,Y 100.08,Z 1159.399,A -85,B 0,C 180,E1 6042.103,E2 6042.103} C_VEL
LIN {X 0,Y 100.444,Z 1168.308,A -85,B 0,C 180,E1 6032.845,E2 6032.845} C_VEL
LIN {X 0,Y 101.015,Z 1172.792,A -85,B 0,C 180,E1 6027.155,E2 6027.155} C_VEL
LIN {X 0,Y 100.418,Z 1177.018,A -85,B 0,C 180,E1 6019.667,E2 6019.667} C_VEL
LIN {X 0,Y 102.189,Z 1182.802,A -85,B 0,C 180,E1 6006.34,E2 6006.34} C_VEL
LIN {X 0,Y 111.551,Z 1187.971,A -85,B 0,C 180,E1 5991.13,E2 5991.13} C_VEL
LIN {X 0,Y 121.504,Z 1190.422,A -85,B 0,C 180,E1 5982.804,E2 5982.804} C_VEL
LIN {X 0,Y 107.082,Z 1182.517,A -85,B 0,C 180,E1 5969.675,E2 5969.675} C_VEL
LIN {X 0,Y 100.399,Z 1174.483,A -85,B 0,C 180,E1 5956.8,E2 5956.8} C_VEL
LIN {X 0,Y 98.479,Z 1168.004,A -85,B 0,C 180,E1 5947.516,E2 5947.516} C_VEL
LIN {X 0,Y 97.374,Z 1165.12,A -85,B 0,C 180,E1 5944.077,E2 5944.077} C_VEL
LIN {X 0,Y 94.299,Z 1160.092,A -85,B 0,C 180,E1 5939.204,E2 5939.204} C_VEL
LIN {X 0,Y 90.446,Z 1152.16,A -85,B 0,C 180,E1 5931.87,E2 5931.87} C_VEL
LIN {X 0,Y 90.285,Z 1149.678,A -85,B 0,C 180,E1 5929.461,E2 5929.461} C_VEL
LIN {X 0,Y 92.515,Z 1137.382,A -85,B 0,C 180,E1 5918.373,E2 5918.373} C_VEL
LIN {X 0,Y 97.081,Z 1123.46,A -85,B 0,C 180,E1 5908.329,E2 5908.329} C_VEL
LIN {X 0,Y 103.511,Z 1108.074,A -85,B 0,C 180,E1 5899.686,E2 5899.686} C_VEL
LIN {X 0,Y 112.028,Z 1089.63,A -85,B 0,C 180,E1 5891.836,E2 5891.836} C_VEL
LIN {X 0,Y 120.832,Z 1070.761,A -85,B 0,C 180,E1 5885.83,E2 5885.83} C_VEL
LIN {X 0,Y 130.312,Z 1049.52,A -85,B 0,C 180,E1 5880.773,E2 5880.773} C_VEL
LIN {X 0,Y 139.408,Z 1027.378,A -85,B 0,C 180,E1 5876.82,E2 5876.82} C_VEL
LIN {X 0,Y 148.012,Z 1003.846,A -85,B 0,C 180,E1 5873.686,E2 5873.686} C_VEL
LIN {X 0,Y 155.98,Z 978.534,A -85,B 0,C 180,E1 5871.164,E2 5871.164} C_VEL
LIN {X 0,Y 162.812,Z 952.353,A -85,B 0,C 180,E1 5869.251,E2 5869.251} C_VEL
LIN {X 0,Y 187.472,Z 834.317,A -85,B 0,C 180,E1 5863.498,E2 5863.498} C_VEL
LIN {X 0,Y 178.995,Z 815.401,A -85,B 0,C 180,E1 5858.194,E2 5858.194} C_VEL
LIN {X 0,Y 171.465,Z 799.321,A -85,B 0,C 180,E1 5852.678,E2 5852.678} C_VEL
LIN {X 0,Y 165.146,Z 786.346,A -85,B 0,C 180,E1 5847.257,E2 5847.257} C_VEL
LIN {X 0,Y 159.395,Z 775.42,A -85,B 0,C 180,E1 5841.528,E2 5841.528} C_VEL
LIN {X 0,Y 157.393,Z 771.829,A -85,B 0,C 180,E1 5839.25,E2 5839.25} C_VEL
LIN {X 0,Y 152.845,Z 776.614,A -85,B 0,C 180,E1 5836.599,E2 5836.599} C_VEL
LIN {X 0,Y 149.16,Z 780.814,A -85,B 0,C 180,E1 5834.232,E2 5834.232} C_VEL
LIN {X 0,Y 145.041,Z 785.915,A -85,B 0,C 180,E1 5831.394,E2 5831.394} C_VEL
LIN {X 0,Y 143.348,Z 788.725,A -85,B 0,C 180,E1 5830.303,E2 5830.303} C_VEL
LIN {X 0,Y 140.003,Z 795.672,A -85,B 0,C 180,E1 5828.514,E2 5828.514} C_VEL
LIN {X 0,Y 129.341,Z 822.682,A -85,B 0,C 180,E1 5823.523,E2 5823.523} C_VEL
LIN {X 0,Y 122.68,Z 839.8,A -85,B 0,C 180,E1 5819.28,E2 5819.28} C_VEL
LIN {X 0,Y 119.976,Z 846.938,A -85,B 0,C 180,E1 5817.028,E2 5817.028} C_VEL
LIN {X 0,Y 108.882,Z 882.399,A -85,B 0,C 180,E1 5809.488,E2 5809.488} C_VEL
LIN {X 0,Y 104.661,Z 897.529,A -85,B 0,C 180,E1 5806.639,E2 5806.639} C_VEL
LIN {X 0,Y 102.865,Z 904.327,A -85,B 0,C 180,E1 5804.522,E2 5804.522} C_VEL
LIN {X 0,Y 102.539,Z 905.91,A -85,B 0,C 180,E1 5803.837,E2 5803.837} C_VEL
LIN {X 0,Y 97.466,Z 985.873,A -85,B 0,C 180,E1 5793.699,E2 5793.699} C_VEL
LIN {X 0,Y 96.057,Z 1023.785,A -85,B 0,C 180,E1 5788.445,E2 5788.445} C_VEL
LIN {X 0,Y 94.975,Z 1041.473,A -85,B 0,C 180,E1 5785.144,E2 5785.144} C_VEL
LIN {X 0,Y 93.896,Z 1058.89,A -85,B 0,C 180,E1 5780.559,E2 5780.559} C_VEL
LIN {X 0,Y 93.188,Z 1074.776,A -85,B 0,C 180,E1 5775.089,E2 5775.089} C_VEL
LIN {X 0,Y 93.155,Z 1089.663,A -85,B 0,C 180,E1 5768.629,E2 5768.629} C_VEL
LIN {X 0,Y 94.149,Z 1103.531,A -85,B 0,C 180,E1 5761.204,E2 5761.204} C_VEL
LIN {X 0,Y 96.854,Z 1116.649,A -85,B 0,C 180,E1 5752.871,E2 5752.871} C_VEL
LIN {X 0,Y 101.864,Z 1128.133,A -85,B 0,C 180,E1 5744.619,E2 5744.619} C_VEL
LIN {X 0,Y 109.519,Z 1138.297,A -85,B 0,C 180,E1 5736.873,E2 5736.873} C_VEL
LIN {X 0,Y 119.927,Z 1146.993,A -85,B 0,C 180,E1 5729.972,E2 5729.972} C_VEL
LIN {X 0,Y 126.876,Z 1151.295,A -85,B 0,C 180,E1 5726.457,E2 5726.457} C_VEL
LIN {X 0,Y 112.585,Z 1148.27,A -85,B 0,C 180,E1 5717.477,E2 5717.477} C_VEL
LIN {X 0,Y 103.029,Z 1143.804,A -85,B 0,C 180,E1 5706.289,E2 5706.289} C_VEL
LIN {X 0,Y 99.651,Z 1139.848,A -85,B 0,C 180,E1 5697.478,E2 5697.478} C_VEL
LIN {X 0,Y 94.63,Z 1147.527,A -85,B 0,C 180,E1 5691.045,E2 5691.045} C_VEL
LIN {X 0,Y 92.4,Z 1157.096,A -85,B 0,C 180,E1 5681.856,E2 5681.856} C_VEL
LIN {X 0,Y 92.86,Z 1165.606,A -85,B 0,C 180,E1 5672.46,E2 5672.46} C_VEL
LIN {X 0,Y 93.534,Z 1169.865,A -85,B 0,C 180,E1 5666.928,E2 5666.928} C_VEL
LIN {X 0,Y 93.012,Z 1173.989,A -85,B 0,C 180,E1 5659.462,E2 5659.462} C_VEL
LIN {X 0,Y 95.229,Z 1180.195,A -85,B 0,C 180,E1 5644.493,E2 5644.493} C_VEL
LIN {X 0,Y 104.627,Z 1185.399,A -85,B 0,C 180,E1 5629.46,E2 5629.46} C_VEL
LIN {X 0,Y 111.976,Z 1187.397,A -85,B 0,C 180,E1 5622.865,E2 5622.865} C_VEL
LIN {X 0,Y 98.411,Z 1179.19,A -85,B 0,C 180,E1 5609.203,E2 5609.203} C_VEL
LIN {X 0,Y 92.31,Z 1170.829,A -85,B 0,C 180,E1 5595.725,E2 5595.725} C_VEL
LIN {X 0,Y 90.615,Z 1163.897,A -85,B 0,C 180,E1 5585.713,E2 5585.713} C_VEL
LIN {X 0,Y 90.075,Z 1157.19,A -85,B 0,C 180,E1 5577.469,E2 5577.469} C_VEL
LIN {X 0,Y 90.285,Z 1149.678,A -85,B 0,C 180,E1 5569.461,E2 5569.461} C_VEL
LIN {X 0,Y 89.99,Z 1145.954,A -85,B 0,C 180,E1 5565.985,E2 5565.985} C_VEL
LIN {X 0,Y 87.997,Z 1139.186,A -85,B 0,C 180,E1 5560.417,E2 5560.417} C_VEL
LIN {X 0,Y 86.588,Z 1131.276,A -85,B 0,C 180,E1 5554.223,E2 5554.223} C_VEL
LIN {X 0,Y 87.252,Z 1127.583,A -85,B 0,C 180,E1 5551.448,E2 5551.448} C_VEL
LIN {X 0,Y 93.422,Z 1112.419,A -85,B 0,C 180,E1 5541.393,E2 5541.393} C_VEL
LIN {X 0,Y 101.816,Z 1094.58,A -85,B 0,C 180,E1 5532.582,E2 5532.582} C_VEL
LIN {X 0,Y 110.927,Z 1075.775,A -85,B 0,C 180,E1 5525.802,E2 5525.802} C_VEL
LIN {X 0,Y 120.497,Z 1055.43,A -85,B 0,C 180,E1 5520.368,E2 5520.368} C_VEL
LIN {X 0,Y 130.136,Z 1033.281,A -85,B 0,C 180,E1 5516.003,E2 5516.003} C_VEL
LIN {X 0,Y 139.239,Z 1009.95,A -85,B 0,C 180,E1 5512.595,E2 5512.595} C_VEL
LIN {X 0,Y 147.758,Z 984.803,A -85,B 0,C 180,E1 5509.872,E2 5509.872} C_VEL
LIN {X 0,Y 154.979,Z 959.097,A -85,B 0,C 180,E1 5507.835,E2 5507.835} C_VEL
LIN {X 0,Y 162.779,Z 924.484,A -85,B 0,C 180,E1 5505.874,E2 5505.874} C_VEL
LIN {X 0,Y 181.433,Z 837.069,A -85,B 0,C 180,E1 5501.77,E2 5501.77} C_VEL
LIN {X 0,Y 173.633,Z 819.099,A -85,B 0,C 180,E1 5496.452,E2 5496.452} C_VEL
LIN {X 0,Y 166.171,Z 802.796,A -85,B 0,C 180,E1 5490.565,E2 5490.565} C_VEL
LIN {X 0,Y 160.687,Z 791.278,A -85,B 0,C 180,E1 5485.454,E2 5485.454} C_VEL
LIN {X 0,Y 155.758,Z 781.554,A -85,B 0,C 180,E1 5480.117,E2 5480.117} C_VEL
LIN {X 0,Y 155.185,Z 780.864,A -85,B 0,C 180,E1 5479.508,E2 5479.508} C_VEL
LIN {X 0,Y 148.805,Z 787.882,A -85,B 0,C 180,E1 5475.762,E2 5475.762} C_VEL
LIN {X 0,Y 144.869,Z 792.604,A -85,B 0,C 180,E1 5473.199,E2 5473.199} C_VEL
LIN {X 0,Y 141.549,Z 798.838,A -85,B 0,C 180,E1 5471.438,E2 5471.438} C_VEL
LIN {X 0,Y 130.218,Z 826.436,A -85,B 0,C 180,E1 5466.618,E2 5466.618} C_VEL
LIN {X 0,Y 123.029,Z 843.976,A -85,B 0,C 180,E1 5462.461,E2 5462.461} C_VEL
LIN {X 0,Y 120.077,Z 851.105,A -85,B 0,C 180,E1 5460.336,E2 5460.336} C_VEL
LIN {X 0,Y 108.729,Z 885.232,A -85,B 0,C 180,E1 5453.446,E2 5453.446} C_VEL
LIN {X 0,Y 104.157,Z 900.552,A -85,B 0,C 180,E1 5450.695,E2 5450.695} C_VEL
LIN {X 0,Y 101.816,Z 908.388,A -85,B 0,C 180,E1 5448.362,E2 5448.362} C_VEL
LIN {X 0,Y 101.249,Z 910.401,A -85,B 0,C 180,E1 5447.874,E2 5447.874} C_VEL
LIN {X 0,Y 95.701,Z 931.048,A -85,B 0,C 180,E1 5444.619,E2 5444.619} C_VEL
LIN {X 0,Y 92.363,Z 944.261,A -85,B 0,C 180,E1 5441.309,E2 5441.309} C_VEL
LIN {X 0,Y 91.193,Z 949.718,A -85,B 0,C 180,E1 5439.025,E2 5439.025} C_VEL
LIN {X 0,Y 91.055,Z 950.907,A -85,B 0,C 180,E1 5438.355,E2 5438.355} C_VEL
LIN {X 0,Y 88.422,Z 1018.409,A -85,B 0,C 180,E1 5428.385,E2 5428.385} C_VEL
LIN {X 0,Y 87.415,Z 1036.733,A -85,B 0,C 180,E1 5425.022,E2 5425.022} C_VEL
LIN {X 0,Y 86.367,Z 1054.681,A -85,B 0,C 180,E1 5420.307,E2 5420.307} C_VEL
LIN {X 0,Y 85.729,Z 1070.234,A -85,B 0,C 180,E1 5414.853,E2 5414.853} C_VEL
LIN {X 0,Y 85.744,Z 1085.663,A -85,B 0,C 180,E1 5408.029,E2 5408.029} C_VEL
LIN {X 0,Y 86.747,Z 1099.173,A -85,B 0,C 180,E1 5400.646,E2 5400.646} C_VEL
LIN {X 0,Y 89.308,Z 1112.244,A -85,B 0,C 180,E1 5392.265,E2 5392.265} C_VEL
LIN {X 0,Y 94.837,Z 1125.317,A -85,B 0,C 180,E1 5382.817,E2 5382.817} C_VEL
LIN {X 0,Y 102.868,Z 1136.088,A -85,B 0,C 180,E1 5374.667,E2 5374.667} C_VEL
LIN {X 0,Y 114.42,Z 1145.927,A -85,B 0,C 180,E1 5367.182,E2 5367.182} C_VEL
LIN {X 0,Y 116.24,Z 1147.224,A -85,B 0,C 180,E1 5366.094,E2 5366.094} C_VEL
LIN {X 0,Y 102.811,Z 1143.176,A -85,B 0,C 180,E1 5356.017,E2 5356.017} C_VEL
LIN {X 0,Y 94.639,Z 1137.605,A -85,B 0,C 180,E1 5343.315,E2 5343.315} C_VEL
LIN {X 0,Y 93.438,Z 1135.859,A -85,B 0,C 180,E1 5339.479,E2 5339.479} C_VEL
LIN {X 0,Y 88.12,Z 1142.957,A -85,B 0,C 180,E1 5333.389,E2 5333.389} C_VEL
LIN {X 0,Y 85.036,Z 1151.462,A -85,B 0,C 180,E1 5324.982,E2 5324.982} C_VEL
LIN {X 0,Y 85.202,Z 1162.328,A -85,B 0,C 180,E1 5312.681,E2 5312.681} C_VEL
LIN {X 0,Y 86.102,Z 1167.268,A -85,B 0,C 180,E1 5305.996,E2 5305.996} C_VEL
LIN {X 0,Y 85.685,Z 1171.961,A -85,B 0,C 180,E1 5296.494,E2 5296.494} C_VEL
LIN {X 0,Y 89.876,Z 1178.713,A -85,B 0,C 180,E1 5278.967,E2 5278.967} C_VEL
LIN {X 0,Y 101.568,Z 1183.751,A -85,B 0,C 180,E1 5264.047,E2 5264.047} C_VEL
LIN {X 0,Y 102.644,Z 1184.04,A -85,B 0,C 180,E1 5263.007,E2 5263.007} C_VEL
LIN {X 0,Y 90.178,Z 1175.806,A -85,B 0,C 180,E1 5249.216,E2 5249.216} C_VEL
LIN {X 0,Y 84.135,Z 1166.466,A -85,B 0,C 180,E1 5233.765,E2 5233.765} C_VEL
LIN {X 0,Y 82.802,Z 1159.912,A -85,B 0,C 180,E1 5224.17,E2 5224.17} C_VEL
LIN {X 0,Y 82.318,Z 1152.065,A -85,B 0,C 180,E1 5214.439,E2 5214.439} C_VEL
LIN {X 0,Y 83.387,Z 1141.469,A -85,B 0,C 180,E1 5203.291,E2 5203.291} C_VEL
LIN {X 0,Y 87.252,Z 1127.583,A -85,B 0,C 180,E1 5191.448,E2 5191.448} C_VEL
LIN {X 0,Y 88.16,Z 1122.482,A -85,B 0,C 180,E1 5187.722,E2 5187.722} C_VEL
LIN {X 0,Y 88.344,Z 1107.363,A -85,B 0,C 180,E1 5177.911,E2 5177.911} C_VEL
LIN {X 0,Y 89.957,Z 1102.448,A -85,B 0,C 180,E1 5175.182,E2 5175.182} C_VEL
LIN {X 0,Y 99.074,Z 1084.353,A -85,B 0,C 180,E1 5167.15,E2 5167.15} C_VEL
LIN {X 0,Y 109.237,Z 1063.983,A -85,B 0,C 180,E1 5160.661,E2 5160.661} C_VEL
LIN {X 0,Y 119.296,Z 1042.469,A -85,B 0,C 180,E1 5155.734,E2 5155.734} C_VEL
LIN {X 0,Y 128.805,Z 1020.035,A -85,B 0,C 180,E1 5151.957,E2 5151.957} C_VEL
LIN {X 0,Y 137.502,Z 996.735,A -85,B 0,C 180,E1 5149.064,E2 5149.064} C_VEL
LIN {X 0,Y 145.362,Z 972.069,A -85,B 0,C 180,E1 5146.798,E2 5146.798} C_VEL
LIN {X 0,Y 152.099,Z 946.278,A -85,B 0,C 180,E1 5145.058,E2 5145.058} C_VEL
LIN {X 0,Y 175.592,Z 839.999,A -85,B 0,C 180,E1 5139.982,E2 5139.982} C_VEL
LIN {X 0,Y 168.638,Z 823.644,A -85,B 0,C 180,E1 5134.92,E2 5134.92} C_VEL
LIN {X 0,Y 161.917,Z 808.334,A -85,B 0,C 180,E1 5129.171,E2 5129.171} C_VEL
LIN {X 0,Y 156.626,Z 796.722,A -85,B 0,C 180,E1 5123.837,E2 5123.837} C_VEL
LIN {X 0,Y 153.186,Z 789.897,A -85,B 0,C 180,E1 5119.94,E2 5119.94} C_VEL
LIN {X 0,Y 148.202,Z 795.307,A -85,B 0,C 180,E1 5117.097,E2 5117.097} C_VEL
LIN {X 0,Y 145.15,Z 798.876,A -85,B 0,C 180,E1 5115.206,E2 5115.206} C_VEL
LIN {X 0,Y 142.362,Z 804.299,A -85,B 0,C 180,E1 5113.983,E2 5113.983} C_VEL
LIN {X 0,Y 130.992,Z 831.041,A -85,B 0,C 180,E1 5109.509,E2 5109.509} C_VEL
LIN {X 0,Y 123.526,Z 848.344,A -85,B 0,C 180,E1 5105.567,E2 5105.567} C_VEL
LIN {X 0,Y 120.567,Z 855.233,A -85,B 0,C 180,E1 5103.636,E2 5103.636} C_VEL
LIN {X 0,Y 109.016,Z 888.062,A -85,B 0,C 180,E1 5097.401,E2 5097.401} C_VEL
LIN {X 0,Y 104.002,Z 903.792,A -85,B 0,C 180,E1 5094.723,E2 5094.723} C_VEL
LIN {X 0,Y 100.949,Z 913.349,A -85,B 0,C 180,E1 5092.156,E2 5092.156} C_VEL
LIN {X 0,Y 94.995,Z 934.024,A -85,B 0,C 180,E1 5089.081,E2 5089.081} C_VEL
LIN {X 0,Y 91.247,Z 947.604,A -85,B 0,C 180,E1 5085.792,E2 5085.792} C_VEL
LIN {X 0,Y 89.469,Z 954.098,A -85,B 0,C 180,E1 5083.178,E2 5083.178} C_VEL
LIN {X 0,Y 84.475,Z 971.673,A -85,B 0,C 180,E1 5079.27,E2 5079.27} C_VEL
LIN {X 0,Y 82.379,Z 979.188,A -85,B 0,C 180,E1 5076.475,E2 5076.475} C_VEL
LIN {X 0,Y 81.615,Z 982.675,A -85,B 0,C 180,E1 5074.283,E2 5074.283} C_VEL
LIN {X 0,Y 81.57,Z 983.955,A -85,B 0,C 180,E1 5073.059,E2 5073.059} C_VEL
LIN {X 0,Y 80.376,Z 1022.244,A -85,B 0,C 180,E1 5066.638,E2 5066.638} C_VEL
LIN {X 0,Y 79.467,Z 1039.391,A -85,B 0,C 180,E1 5062.941,E2 5062.941} C_VEL
LIN {X 0,Y 78.614,Z 1056.648,A -85,B 0,C 180,E1 5057.756,E2 5057.756} C_VEL
LIN {X 0,Y 78.259,Z 1073.484,A -85,B 0,C 180,E1 5051.033,E2 5051.033} C_VEL
LIN {X 0,Y 78.822,Z 1088.129,A -85,B 0,C 180,E1 5043.621,E2 5043.621} C_VEL
LIN {X 0,Y 80.693,Z 1102.241,A -85,B 0,C 180,E1 5035.009,E2 5035.009} C_VEL
LIN {X 0,Y 84.737,Z 1115.579,A -85,B 0,C 180,E1 5025.638,E2 5025.638} C_VEL
LIN {X 0,Y 91.92,Z 1128.147,A -85,B 0,C 180,E1 5016.252,E2 5016.252} C_VEL
LIN {X 0,Y 102.185,Z 1139.092,A -85,B 0,C 180,E1 5008.089,E2 5008.089} C_VEL
LIN {X 0,Y 106.135,Z 1142.374,A -85,B 0,C 180,E1 5005.601,E2 5005.601} C_VEL
LIN {X 0,Y 93.792,Z 1137.426,A -85,B 0,C 180,E1 4994.399,E2 4994.399} C_VEL
LIN {X 0,Y 87.367,Z 1131.859,A -85,B 0,C 180,E1 4981.755,E2 4981.755} C_VEL
LIN {X 0,Y 81.036,Z 1139.675,A -85,B 0,C 180,E1 4974.793,E2 4974.793} C_VEL
LIN {X 0,Y 77.428,Z 1148.898,A -85,B 0,C 180,E1 4964.957,E2 4964.957} C_VEL
LIN {X 0,Y 77.576,Z 1158.813,A -85,B 0,C 180,E1 4952.945,E2 4952.945} C_VEL
LIN {X 0,Y 78.761,Z 1164.47,A -85,B 0,C 180,E1 4944.892,E2 4944.892} C_VEL
LIN {X 0,Y 78.511,Z 1169.23,A -85,B 0,C 180,E1 4934.477,E2 4934.477} C_VEL
LIN {X 0,Y 82.69,Z 1175.375,A -85,B 0,C 180,E1 4917.845,E2 4917.845} C_VEL
LIN {X 0,Y 93.472,Z 1180.35,A -85,B 0,C 180,E1 4903.223,E2 4903.223} C_VEL
LIN {X 0,Y 81.295,Z 1171.358,A -85,B 0,C 180,E1 4887.881,E2 4887.881} C_VEL
LIN {X 0,Y 76.172,Z 1162.206,A -85,B 0,C 180,E1 4872.14,E2 4872.14} C_VEL
LIN {X 0,Y 74.977,Z 1155.604,A -85,B 0,C 180,E1 4862.309,E2 4862.309} C_VEL
LIN {X 0,Y 74.72,Z 1146.455,A -85,B 0,C 180,E1 4850.776,E2 4850.776} C_VEL
LIN {X 0,Y 76.652,Z 1134.946,A -85,B 0,C 180,E1 4838.595,E2 4838.595} C_VEL
LIN {X 0,Y 81.65,Z 1120.493,A -85,B 0,C 180,E1 4826.397,E2 4826.397} C_VEL
LIN {X 0,Y 89.196,Z 1104.023,A -85,B 0,C 180,E1 4815.991,E2 4815.991} C_VEL
LIN {X 0,Y 89.957,Z 1102.448,A -85,B 0,C 180,E1 4815.182,E2 4815.182} C_VEL
LIN {X 0,Y 91.841,Z 1096.713,A -85,B 0,C 180,E1 4812.196,E2 4812.196} C_VEL
LIN {X 0,Y 94.302,Z 1080.166,A -85,B 0,C 180,E1 4804.068,E2 4804.068} C_VEL
LIN {X 0,Y 96.423,Z 1074.771,A -85,B 0,C 180,E1 4801.978,E2 4801.978} C_VEL
LIN {X 0,Y 107.135,Z 1053.575,A -85,B 0,C 180,E1 4796.025,E2 4796.025} C_VEL
LIN {X 0,Y 117.237,Z 1031.844,A -85,B 0,C 180,E1 4791.653,E2 4791.653} C_VEL
LIN {X 0,Y 126.855,Z 1008.536,A -85,B 0,C 180,E1 4788.267,E2 4788.267} C_VEL
LIN {X 0,Y 135.509,Z 984.301,A -85,B 0,C 180,E1 4785.689,E2 4785.689} C_VEL
LIN {X 0,Y 142.987,Z 959.249,A -85,B 0,C 180,E1 4783.726,E2 4783.726} C_VEL
LIN {X 0,Y 151.393,Z 923.937,A -85,B 0,C 180,E1 4781.773,E2 4781.773} C_VEL
LIN {X 0,Y 169.774,Z 842.721,A -85,B 0,C 180,E1 4778.024,E2 4778.024} C_VEL
LIN {X 0,Y 163.007,Z 826.408,A -85,B 0,C 180,E1 4772.659,E2 4772.659} C_VEL
LIN {X 0,Y 156.875,Z 811.944,A -85,B 0,C 180,E1 4766.899,E2 4766.899} C_VEL
LIN {X 0,Y 152.193,Z 801.354,A -85,B 0,C 180,E1 4761.695,E2 4761.695} C_VEL
LIN {X 0,Y 151.054,Z 798.94,A -85,B 0,C 180,E1 4760.288,E2 4760.288} C_VEL
LIN {X 0,Y 145.888,Z 804.748,A -85,B 0,C 180,E1 4757.428,E2 4757.428} C_VEL
LIN {X 0,Y 143.862,Z 808.774,A -85,B 0,C 180,E1 4756.624,E2 4756.624} C_VEL
LIN {X 0,Y 131.837,Z 836.18,A -85,B 0,C 180,E1 4752.261,E2 4752.261} C_VEL
LIN {X 0,Y 124.022,Z 853.485,A -85,B 0,C 180,E1 4748.432,E2 4748.432} C_VEL
LIN {X 0,Y 121.416,Z 859.179,A -85,B 0,C 180,E1 4746.94,E2 4746.94} C_VEL
LIN {X 0,Y 109.724,Z 890.795,A -85,B 0,C 180,E1 4741.337,E2 4741.337} C_VEL
LIN {X 0,Y 104.389,Z 906.832,A -85,B 0,C 180,E1 4738.788,E2 4738.788} C_VEL
LIN {X 0,Y 101.005,Z 916.488,A -85,B 0,C 180,E1 4736.426,E2 4736.426} C_VEL
LIN {X 0,Y 94.805,Z 937.047,A -85,B 0,C 180,E1 4733.572,E2 4733.572} C_VEL
LIN {X 0,Y 90.568,Z 950.796,A -85,B 0,C 180,E1 4730.397,E2 4730.397} C_VEL
LIN {X 0,Y 88.082,Z 958.772,A -85,B 0,C 180,E1 4727.588,E2 4727.588} C_VEL
LIN {X 0,Y 83.37,Z 973.652,A -85,B 0,C 180,E1 4724.534,E2 4724.534} C_VEL
LIN {X 0,Y 80.3,Z 982.841,A -85,B 0,C 180,E1 4721.275,E2 4721.275} C_VEL
LIN {X 0,Y 78.818,Z 988.076,A -85,B 0,C 180,E1 4717.997,E2 4717.997} C_VEL
LIN {X 0,Y 74.931,Z 999.766,A -85,B 0,C 180,E1 4714.194,E2 4714.194} C_VEL
LIN {X 0,Y 73.332,Z 1005.259,A -85,B 0,C 180,E1 4711.186,E2 4711.186} C_VEL
LIN {X 0,Y 72.949,Z 1008.02,A -85,B 0,C 180,E1 4708.648,E2 4708.648} C_VEL
LIN {X 0,Y 73.057,Z 1008.758,A -85,B 0,C 180,E1 4707.74,E2 4707.74} C_VEL
LIN {X 0,Y 72.052,Z 1033.485,A -85,B 0,C 180,E1 4702.631,E2 4702.631} C_VEL
LIN {X 0,Y 71.277,Z 1050.747,A -85,B 0,C 180,E1 4697.502,E2 4697.502} C_VEL
LIN {X 0,Y 70.988,Z 1067.019,A -85,B 0,C 180,E1 4690.944,E2 4690.944} C_VEL
LIN {X 0,Y 71.547,Z 1082.35,A -85,B 0,C 180,E1 4683.187,E2 4683.187} C_VEL
LIN {X 0,Y 73.379,Z 1096.344,A -85,B 0,C 180,E1 4674.51,E2 4674.51} C_VEL
LIN {X 0,Y 77.161,Z 1109.85,A -85,B 0,C 180,E1 4664.963,E2 4664.963} C_VEL
LIN {X 0,Y 83.909,Z 1122.658,A -85,B 0,C 180,E1 4655.334,E2 4655.334} C_VEL
LIN {X 0,Y 93.561,Z 1134.103,A -85,B 0,C 180,E1 4646.958,E2 4646.958} C_VEL
LIN {X 0,Y 96.479,Z 1136.791,A -85,B 0,C 180,E1 4644.944,E2 4644.944} C_VEL
LIN {X 0,Y 85.375,Z 1131.04,A -85,B 0,C 180,E1 4632.432,E2 4632.432} C_VEL
LIN {X 0,Y 81.779,Z 1127.466,A -85,B 0,C 180,E1 4624.424,E2 4624.424} C_VEL
LIN {X 0,Y 75.522,Z 1134.142,A -85,B 0,C 180,E1 4618.453,E2 4618.453} C_VEL
LIN {X 0,Y 70.724,Z 1142.877,A -85,B 0,C 180,E1 4608.964,E2 4608.964} C_VEL
LIN {X 0,Y 69.946,Z 1155.174,A -85,B 0,C 180,E1 4593.267,E2 4593.267} C_VEL
LIN {X 0,Y 71.443,Z 1161.4,A -85,B 0,C 180,E1 4583.963,E2 4583.963} C_VEL
LIN {X 0,Y 71.562,Z 1166.736,A -85,B 0,C 180,E1 4571.243,E2 4571.243} C_VEL
LIN {X 0,Y 78.42,Z 1173.592,A -85,B 0,C 180,E1 4551.323,E2 4551.323} C_VEL
LIN {X 0,Y 84.375,Z 1176.262,A -85,B 0,C 180,E1 4543.438,E2 4543.438} C_VEL
LIN {X 0,Y 72.534,Z 1166.511,A -85,B 0,C 180,E1 4526.194,E2 4526.194} C_VEL
LIN {X 0,Y 68.688,Z 1158.93,A -85,B 0,C 180,E1 4512.631,E2 4512.631} C_VEL
LIN {X 0,Y 67.388,Z 1152.579,A -85,B 0,C 180,E1 4502.57,E2 4502.57} C_VEL
LIN {X 0,Y 67.054,Z 1143.779,A -85,B 0,C 180,E1 4490.578,E2 4490.578} C_VEL
LIN {X 0,Y 69.415,Z 1131.216,A -85,B 0,C 180,E1 4476.234,E2 4476.234} C_VEL
LIN {X 0,Y 75.111,Z 1116.342,A -85,B 0,C 180,E1 4463.22,E2 4463.22} C_VEL
LIN {X 0,Y 83.384,Z 1099.479,A -85,B 0,C 180,E1 4452.507,E2 4452.507} C_VEL
LIN {X 0,Y 93.433,Z 1080.411,A -85,B 0,C 180,E1 4443.991,E2 4443.991} C_VEL
LIN {X 0,Y 96.423,Z 1074.771,A -85,B 0,C 180,E1 4441.978,E2 4441.978} C_VEL
LIN {X 0,Y 98.797,Z 1068.485,A -85,B 0,C 180,E1 4439.698,E2 4439.698} C_VEL
LIN {X 0,Y 102.225,Z 1050.803,A -85,B 0,C 180,E1 4433.288,E2 4433.288} C_VEL
LIN {X 0,Y 104.409,Z 1045.018,A -85,B 0,C 180,E1 4431.803,E2 4431.803} C_VEL
LIN {X 0,Y 114.508,Z 1023.096,A -85,B 0,C 180,E1 4427.902,E2 4427.902} C_VEL
LIN {X 0,Y 124.114,Z 999.432,A -85,B 0,C 180,E1 4424.861,E2 4424.861} C_VEL
LIN {X 0,Y 132.636,Z 974.695,A -85,B 0,C 180,E1 4422.561,E2 4422.561} C_VEL
LIN {X 0,Y 140.185,Z 947.873,A -85,B 0,C 180,E1 4420.782,E2 4420.782} C_VEL
LIN {X 0,Y 164.085,Z 845.655,A -85,B 0,C 180,E1 4416.03,E2 4416.03} C_VEL
LIN {X 0,Y 157.932,Z 830.181,A -85,B 0,C 180,E1 4410.649,E2 4410.649} C_VEL
LIN {X 0,Y 152.232,Z 816.097,A -85,B 0,C 180,E1 4404.729,E2 4404.729} C_VEL
LIN {X 0,Y 148.911,Z 808.254,A -85,B 0,C 180,E1 4400.713,E2 4400.713} C_VEL
LIN {X 0,Y 146.748,Z 810.707,A -85,B 0,C 180,E1 4399.593,E2 4399.593} C_VEL
LIN {X 0,Y 132.927,Z 841.2,A -85,B 0,C 180,E1 4395.003,E2 4395.003} C_VEL
LIN {X 0,Y 124.866,Z 858.284,A -85,B 0,C 180,E1 4391.366,E2 4391.366} C_VEL
LIN {X 0,Y 122.543,Z 863.28,A -85,B 0,C 180,E1 4390.169,E2 4390.169} C_VEL
LIN {X 0,Y 110.876,Z 893.583,A -85,B 0,C 180,E1 4385.203,E2 4385.203} C_VEL
LIN {X 0,Y 105.182,Z 909.777,A -85,B 0,C 180,E1 4382.833,E2 4382.833} C_VEL
LIN {X 0,Y 101.607,Z 919.495,A -85,B 0,C 180,E1 4380.68,E2 4380.68} C_VEL
LIN {X 0,Y 95.107,Z 940.007,A -85,B 0,C 180,E1 4378.071,E2 4378.071} C_VEL
LIN {X 0,Y 90.406,Z 953.994,A -85,B 0,C 180,E1 4375.041,E2 4375.041} C_VEL
LIN {X 0,Y 87.599,Z 961.935,A -85,B 0,C 180,E1 4372.47,E2 4372.47} C_VEL
LIN {X 0,Y 82.537,Z 976.278,A -85,B 0,C 180,E1 4369.723,E2 4369.723} C_VEL
LIN {X 0,Y 79.052,Z 985.704,A -85,B 0,C 180,E1 4366.636,E2 4366.636} C_VEL
LIN {X 0,Y 76.376,Z 992.79,A -85,B 0,C 180,E1 4362.88,E2 4362.88} C_VEL
LIN {X 0,Y 72.391,Z 1003.317,A -85,B 0,C 180,E1 4359.424,E2 4359.424} C_VEL
LIN {X 0,Y 70.163,Z 1009.956,A -85,B 0,C 180,E1 4355.699,E2 4355.699} C_VEL
LIN {X 0,Y 69.269,Z 1013.293,A -85,B 0,C 180,E1 4352.751,E2 4352.751} C_VEL
LIN {X 0,Y 65.797,Z 1022.996,A -85,B 0,C 180,E1 4348.578,E2 4348.578} C_VEL
LIN {X 0,Y 64.387,Z 1028.267,A -85,B 0,C 180,E1 4344.768,E2 4344.768} C_VEL
LIN {X 0,Y 64.337,Z 1030.609,A -85,B 0,C 180,E1 4341.879,E2 4341.879} C_VEL
LIN {X 0,Y 64.522,Z 1031.239,A -85,B 0,C 180,E1 4340.994,E2 4340.994} C_VEL
LIN {X 0,Y 63.945,Z 1047.462,A -85,B 0,C 180,E1 4335.861,E2 4335.861} C_VEL
LIN {X 0,Y 63.834,Z 1064.696,A -85,B 0,C 180,E1 4328.538,E2 4328.538} C_VEL
LIN {X 0,Y 64.816,Z 1080.305,A -85,B 0,C 180,E1 4319.981,E2 4319.981} C_VEL
LIN {X 0,Y 67.032,Z 1094.119,A -85,B 0,C 180,E1 4310.97,E2 4310.97} C_VEL
LIN {X 0,Y 71.33,Z 1107.416,A -85,B 0,C 180,E1 4301.173,E2 4301.173} C_VEL
LIN {X 0,Y 78.863,Z 1120.668,A -85,B 0,C 180,E1 4291.18,E2 4291.18} C_VEL
LIN {X 0,Y 87.289,Z 1130.545,A -85,B 0,C 180,E1 4284.025,E2 4284.025} C_VEL
LIN {X 0,Y 77.269,Z 1123.708,A -85,B 0,C 180,E1 4269.338,E2 4269.338} C_VEL
LIN {X 0,Y 76.424,Z 1123.037,A -85,B 0,C 180,E1 4267.459,E2 4267.459} C_VEL
LIN {X 0,Y 69.358,Z 1129.907,A -85,B 0,C 180,E1 4261.25,E2 4261.25} C_VEL
LIN {X 0,Y 63.484,Z 1139.392,A -85,B 0,C 180,E1 4250.26,E2 4250.26} C_VEL
LIN {X 0,Y 62.24,Z 1150.474,A -85,B 0,C 180,E1 4234.89,E2 4234.89} C_VEL
LIN {X 0,Y 64.162,Z 1158.135,A -85,B 0,C 180,E1 4222.826,E2 4222.826} C_VEL
LIN {X 0,Y 64.373,Z 1162.458,A -85,B 0,C 180,E1 4211.889,E2 4211.889} C_VEL
LIN {X 0,Y 69.655,Z 1168.794,A -85,B 0,C 180,E1 4192.908,E2 4192.908} C_VEL
LIN {X 0,Y 75.516,Z 1171.803,A -85,B 0,C 180,E1 4183.796,E2 4183.796} C_VEL
LIN {X 0,Y 64.177,Z 1161.692,A -85,B 0,C 180,E1 4164.897,E2 4164.897} C_VEL
LIN {X 0,Y 60.779,Z 1153.974,A -85,B 0,C 180,E1 4150.446,E2 4150.446} C_VEL
LIN {X 0,Y 59.44,Z 1146.341,A -85,B 0,C 180,E1 4138.093,E2 4138.093} C_VEL
LIN {X 0,Y 60.046,Z 1135.877,A -85,B 0,C 180,E1 4123.578,E2 4123.578} C_VEL
LIN {X 0,Y 64.298,Z 1121.998,A -85,B 0,C 180,E1 4108.104,E2 4108.104} C_VEL
LIN {X 0,Y 71.25,Z 1107.228,A -85,B 0,C 180,E1 4096.026,E2 4096.026} C_VEL
LIN {X 0,Y 80.83,Z 1089.522,A -85,B 0,C 180,E1 4085.907,E2 4085.907} C_VEL
LIN {X 0,Y 91.822,Z 1069.458,A -85,B 0,C 180,E1 4078.142,E2 4078.142} C_VEL
LIN {X 0,Y 102.797,Z 1048.308,A -85,B 0,C 180,E1 4072.509,E2 4072.509} C_VEL
LIN {X 0,Y 104.409,Z 1045.018,A -85,B 0,C 180,E1 4071.803,E2 4071.803} C_VEL
LIN {X 0,Y 106.821,Z 1038.335,A -85,B 0,C 180,E1 4070.148,E2 4070.148} C_VEL
LIN {X 0,Y 110.341,Z 1019.724,A -85,B 0,C 180,E1 4065.044,E2 4065.044} C_VEL
LIN {X 0,Y 112.355,Z 1013.653,A -85,B 0,C 180,E1 4063.981,E2 4063.981} C_VEL
LIN {X 0,Y 121.576,Z 990.196,A -85,B 0,C 180,E1 4061.39,E2 4061.39} C_VEL
LIN {X 0,Y 129.842,Z 965.23,A -85,B 0,C 180,E1 4059.398,E2 4059.398} C_VEL
LIN {X 0,Y 137.205,Z 937.662,A -85,B 0,C 180,E1 4057.819,E2 4057.819} C_VEL
LIN {X 0,Y 158.504,Z 848.393,A -85,B 0,C 180,E1 4053.848,E2 4053.848} C_VEL
LIN {X 0,Y 152.392,Z 832.474,A -85,B 0,C 180,E1 4047.937,E2 4047.937} C_VEL
LIN {X 0,Y 147.418,Z 819.625,A -85,B 0,C 180,E1 4042.101,E2 4042.101} C_VEL
LIN {X 0,Y 146.977,Z 818.917,A -85,B 0,C 180,E1 4041.61,E2 4041.61} C_VEL
LIN {X 0,Y 134.191,Z 846.463,A -85,B 0,C 180,E1 4037.65,E2 4037.65} C_VEL
LIN {X 0,Y 125.763,Z 863.615,A -85,B 0,C 180,E1 4034.119,E2 4034.119} C_VEL
LIN {X 0,Y 123.974,Z 867.423,A -85,B 0,C 180,E1 4033.348,E2 4033.348} C_VEL
LIN {X 0,Y 112.432,Z 896.26,A -85,B 0,C 180,E1 4029,E2 4029} C_VEL
LIN {X 0,Y 106.43,Z 912.76,A -85,B 0,C 180,E1 4026.796,E2 4026.796} C_VEL
LIN {X 0,Y 102.739,Z 922.294,A -85,B 0,C 180,E1 4024.889,E2 4024.889} C_VEL
LIN {X 0,Y 95.962,Z 942.805,A -85,B 0,C 180,E1 4022.546,E2 4022.546} C_VEL
LIN {X 0,Y 90.716,Z 957.306,A -85,B 0,C 180,E1 4019.646,E2 4019.646} C_VEL
LIN {X 0,Y 87.759,Z 964.577,A -85,B 0,C 180,E1 4017.443,E2 4017.443} C_VEL
LIN {X 0,Y 82.37,Z 978.821,A -85,B 0,C 180,E1 4014.995,E2 4014.995} C_VEL
LIN {X 0,Y 78.099,Z 988.996,A -85,B 0,C 180,E1 4011.914,E2 4011.914} C_VEL
LIN {X 0,Y 74.918,Z 996.343,A -85,B 0,C 180,E1 4008.339,E2 4008.339} C_VEL
LIN {X 0,Y 70.562,Z 1006.6,A -85,B 0,C 180,E1 4005.088,E2 4005.088} C_VEL
LIN {X 0,Y 67.532,Z 1013.819,A -85,B 0,C 180,E1 4001.132,E2 4001.132} C_VEL
LIN {X 0,Y 66.137,Z 1017.52,A -85,B 0,C 180,E1 3998.281,E2 3998.281} C_VEL
LIN {X 0,Y 62.344,Z 1026.772,A -85,B 0,C 180,E1 3994.123,E2 3994.123} C_VEL
LIN {X 0,Y 60.255,Z 1033.046,A -85,B 0,C 180,E1 3989.286,E2 3989.286} C_VEL
LIN {X 0,Y 59.623,Z 1036.218,A -85,B 0,C 180,E1 3985.827,E2 3985.827} C_VEL
LIN {X 0,Y 56.746,Z 1044.946,A -85,B 0,C 180,E1 3980.072,E2 3980.072} C_VEL
LIN {X 0,Y 55.877,Z 1050.484,A -85,B 0,C 180,E1 3974.485,E2 3974.485} C_VEL
LIN {X 0,Y 56.535,Z 1053.254,A -85,B 0,C 180,E1 3970.165,E2 3970.165} C_VEL
LIN {X 0,Y 56.711,Z 1053.64,A -85,B 0,C 180,E1 3969.619,E2 3969.619} C_VEL
LIN {X 0,Y 57.465,Z 1070.12,A -85,B 0,C 180,E1 3960.975,E2 3960.975} C_VEL
LIN {X 0,Y 59.316,Z 1083.877,A -85,B 0,C 180,E1 3952.229,E2 3952.229} C_VEL
LIN {X 0,Y 63.023,Z 1097.773,A -85,B 0,C 180,E1 3942.118,E2 3942.118} C_VEL
LIN {X 0,Y 70.11,Z 1112.405,A -85,B 0,C 180,E1 3930.975,E2 3930.975} C_VEL
LIN {X 0,Y 78.696,Z 1123.683,A -85,B 0,C 180,E1 3922.813,E2 3922.813} C_VEL
LIN {X 0,Y 71.664,Z 1118.241,A -85,B 0,C 180,E1 3910.962,E2 3910.962} C_VEL
LIN {X 0,Y 64.808,Z 1124.087,A -85,B 0,C 180,E1 3905.878,E2 3905.878} C_VEL
LIN {X 0,Y 57.785,Z 1132.976,A -85,B 0,C 180,E1 3895.617,E2 3895.617} C_VEL
LIN {X 0,Y 54.56,Z 1142.576,A -85,B 0,C 180,E1 3881.615,E2 3881.615} C_VEL
LIN {X 0,Y 56.35,Z 1153.372,A -85,B 0,C 180,E1 3863.875,E2 3863.875} C_VEL
LIN {X 0,Y 57.137,Z 1155.432,A -85,B 0,C 180,E1 3859.908,E2 3859.908} C_VEL
LIN {X 0,Y 58.969,Z 1161.556,A -85,B 0,C 180,E1 3841.641,E2 3841.641} C_VEL
LIN {X 0,Y 66.741,Z 1166.976,A -85,B 0,C 180,E1 3824.184,E2 3824.184} C_VEL
LIN {X 0,Y 56.187,Z 1156.975,A -85,B 0,C 180,E1 3804.185,E2 3804.185} C_VEL
LIN {X 0,Y 53.274,Z 1150.286,A -85,B 0,C 180,E1 3790.841,E2 3790.841} C_VEL
LIN {X 0,Y 51.779,Z 1142.202,A -85,B 0,C 180,E1 3776.703,E2 3776.703} C_VEL
LIN {X 0,Y 53.059,Z 1130.386,A -85,B 0,C 180,E1 3759.045,E2 3759.045} C_VEL
LIN {X 0,Y 58.248,Z 1116.618,A -85,B 0,C 180,E1 3743.099,E2 3743.099} C_VEL
LIN {X 0,Y 66.85,Z 1100.308,A -85,B 0,C 180,E1 3730.042,E2 3730.042} C_VEL
LIN {X 0,Y 77.551,Z 1081.81,A -85,B 0,C 180,E1 3720.282,E2 3720.282} C_VEL
LIN {X 0,Y 88.744,Z 1062.06,A -85,B 0,C 180,E1 3713.364,E2 3713.364} C_VEL
LIN {X 0,Y 100.005,Z 1040.505,A -85,B 0,C 180,E1 3708.267,E2 3708.267} C_VEL
LIN {X 0,Y 110.505,Z 1018.002,A -85,B 0,C 180,E1 3704.544,E2 3704.544} C_VEL
LIN {X 0,Y 112.355,Z 1013.653,A -85,B 0,C 180,E1 3703.981,E2 3703.981} C_VEL
LIN {X 0,Y 114.536,Z 1006.719,A -85,B 0,C 180,E1 3702.777,E2 3702.777} C_VEL
LIN {X 0,Y 117.527,Z 987.268,A -85,B 0,C 180,E1 3698.641,E2 3698.641} C_VEL
LIN {X 0,Y 119.22,Z 981.013,A -85,B 0,C 180,E1 3697.864,E2 3697.864} C_VEL
LIN {X 0,Y 127.266,Z 955.458,A -85,B 0,C 180,E1 3696.142,E2 3696.142} C_VEL
LIN {X 0,Y 146.922,Z 876.822,A -85,B 0,C 180,E1 3692.595,E2 3692.595} C_VEL
LIN {X 0,Y 153.139,Z 851.4,A -85,B 0,C 180,E1 3691.604,E2 3691.604} C_VEL
LIN {X 0,Y 147.329,Z 835.54,A -85,B 0,C 180,E1 3685.334,E2 3685.334} C_VEL
LIN {X 0,Y 145.534,Z 831.101,A -85,B 0,C 180,E1 3683.196,E2 3683.196} C_VEL
LIN {X 0,Y 132.473,Z 858.142,A -85,B 0,C 180,E1 3679.129,E2 3679.129} C_VEL
LIN {X 0,Y 126.04,Z 870.725,A -85,B 0,C 180,E1 3676.558,E2 3676.558} C_VEL
LIN {X 0,Y 114.35,Z 899.077,A -85,B 0,C 180,E1 3672.676,E2 3672.676} C_VEL
LIN {X 0,Y 108.007,Z 915.932,A -85,B 0,C 180,E1 3670.632,E2 3670.632} C_VEL
LIN {X 0,Y 104.329,Z 925.001,A -85,B 0,C 180,E1 3669.005,E2 3669.005} C_VEL
LIN {X 0,Y 97.319,Z 945.635,A -85,B 0,C 180,E1 3666.92,E2 3666.92} C_VEL
LIN {X 0,Y 91.553,Z 960.394,A -85,B 0,C 180,E1 3664.258,E2 3664.258} C_VEL
LIN {X 0,Y 88.563,Z 967.103,A -85,B 0,C 180,E1 3662.377,E2 3662.377} C_VEL
LIN {X 0,Y 82.45,Z 982.155,A -85,B 0,C 180,E1 3660.091,E2 3660.091} C_VEL
LIN {X 0,Y 77.435,Z 992.919,A -85,B 0,C 180,E1 3657.037,E2 3657.037} C_VEL
LIN {X 0,Y 74.129,Z 999.641,A -85,B 0,C 180,E1 3653.999,E2 3653.999} C_VEL
LIN {X 0,Y 69.043,Z 1010.44,A -85,B 0,C 180,E1 3650.756,E2 3650.756} C_VEL
LIN {X 0,Y 65.033,Z 1018.653,A -85,B 0,C 180,E1 3646.243,E2 3646.243} C_VEL
LIN {X 0,Y 64.077,Z 1020.75,A -85,B 0,C 180,E1 3644.575,E2 3644.575} C_VEL
LIN {X 0,Y 59.487,Z 1030.384,A -85,B 0,C 180,E1 3640.297,E2 3640.297} C_VEL
LIN {X 0,Y 56.627,Z 1037.2,A -85,B 0,C 180,E1 3634.992,E2 3634.992} C_VEL
LIN {X 0,Y 55.721,Z 1039.926,A -85,B 0,C 180,E1 3631.936,E2 3631.936} C_VEL
LIN {X 0,Y 52.311,Z 1048.416,A -85,B 0,C 180,E1 3626.053,E2 3626.053} C_VEL
LIN {X 0,Y 50.754,Z 1054.513,A -85,B 0,C 180,E1 3619.541,E2 3619.541} C_VEL
LIN {X 0,Y 50.844,Z 1058.411,A -85,B 0,C 180,E1 3613.625,E2 3613.625} C_VEL
LIN {X 0,Y 49.34,Z 1067.268,A -85,B 0,C 180,E1 3604.624,E2 3604.624} C_VEL
LIN {X 0,Y 50.11,Z 1073.463,A -85,B 0,C 180,E1 3596.543,E2 3596.543} C_VEL
LIN {X 0,Y 52.565,Z 1077.488,A -85,B 0,C 180,E1 3590.119,E2 3590.119} C_VEL
LIN {X 0,Y 56.899,Z 1092.494,A -85,B 0,C 180,E1 3578.862,E2 3578.862} C_VEL
LIN {X 0,Y 63.934,Z 1106.891,A -85,B 0,C 180,E1 3567.855,E2 3567.855} C_VEL
LIN {X 0,Y 70.621,Z 1116.227,A -85,B 0,C 180,E1 3561.124,E2 3561.124} C_VEL
LIN {X 0,Y 67.253,Z 1113.389,A -85,B 0,C 180,E1 3554.91,E2 3554.91} C_VEL
LIN {X 0,Y 59.405,Z 1119.523,A -85,B 0,C 180,E1 3549.744,E2 3549.744} C_VEL
LIN {X 0,Y 50.956,Z 1129.224,A -85,B 0,C 180,E1 3538.078,E2 3538.078} C_VEL
LIN {X 0,Y 47.097,Z 1139.606,A -85,B 0,C 180,E1 3520.998,E2 3520.998} C_VEL
LIN {X 0,Y 49.189,Z 1149.986,A -85,B 0,C 180,E1 3501.803,E2 3501.803} C_VEL
LIN {X 0,Y 50.134,Z 1152.212,A -85,B 0,C 180,E1 3497.311,E2 3497.311} C_VEL
LIN {X 0,Y 54.067,Z 1159.293,A -85,B 0,C 180,E1 3473.698,E2 3473.698} C_VEL
LIN {X 0,Y 58.18,Z 1161.871,A -85,B 0,C 180,E1 3464.829,E2 3464.829} C_VEL
LIN {X 0,Y 48.886,Z 1152.796,A -85,B 0,C 180,E1 3445.465,E2 3445.465} C_VEL
LIN {X 0,Y 46.002,Z 1146.888,A -85,B 0,C 180,E1 3432.581,E2 3432.581} C_VEL
LIN {X 0,Y 44.207,Z 1138.455,A -85,B 0,C 180,E1 3416.137,E2 3416.137} C_VEL
LIN {X 0,Y 45.936,Z 1126.202,A -85,B 0,C 180,E1 3395.601,E2 3395.601} C_VEL
LIN {X 0,Y 52.76,Z 1110.835,A -85,B 0,C 180,E1 3377.013,E2 3377.013} C_VEL
LIN {X 0,Y 62.639,Z 1093.979,A -85,B 0,C 180,E1 3363.932,E2 3363.932} C_VEL
LIN {X 0,Y 74.382,Z 1074.779,A -85,B 0,C 180,E1 3354.639,E2 3354.639} C_VEL
LIN {X 0,Y 86.615,Z 1053.55,A -85,B 0,C 180,E1 3348.17,E2 3348.17} C_VEL
LIN {X 0,Y 98.245,Z 1031.201,A -85,B 0,C 180,E1 3343.66,E2 3343.66} C_VEL
LIN {X 0,Y 109.197,Z 1007.054,A -85,B 0,C 180,E1 3340.35,E2 3340.35} C_VEL
LIN {X 0,Y 119.091,Z 981.391,A -85,B 0,C 180,E1 3337.893,E2 3337.893} C_VEL
LIN {X 0,Y 119.22,Z 981.013,A -85,B 0,C 180,E1 3337.864,E2 3337.864} C_VEL
LIN {X 0,Y 121.022,Z 973.684,A -85,B 0,C 180,E1 3336.984,E2 3336.984} C_VEL
LIN {X 0,Y 122.101,Z 963.268,A -85,B 0,C 180,E1 3335.124,E2 3335.124} C_VEL
LIN {X 0,Y 123.38,Z 951.673,A -85,B 0,C 180,E1 3333.302,E2 3333.302} C_VEL
LIN {X 0,Y 124.285,Z 947.393,A -85,B 0,C 180,E1 3332.953,E2 3332.953} C_VEL
LIN {X 0,Y 147.831,Z 854.273,A -85,B 0,C 180,E1 3329.182,E2 3329.182} C_VEL
LIN {X 0,Y 143.975,Z 843.517,A -85,B 0,C 180,E1 3324.695,E2 3324.695} C_VEL
LIN {X 0,Y 132.869,Z 865.609,A -85,B 0,C 180,E1 3321.324,E2 3321.324} C_VEL
LIN {X 0,Y 128.263,Z 874.419,A -85,B 0,C 180,E1 3319.623,E2 3319.623} C_VEL
LIN {X 0,Y 116.69,Z 901.81,A -85,B 0,C 180,E1 3316.234,E2 3316.234} C_VEL
LIN {X 0,Y 110.027,Z 918.936,A -85,B 0,C 180,E1 3314.382,E2 3314.382} C_VEL
LIN {X 0,Y 106.373,Z 927.779,A -85,B 0,C 180,E1 3312.981,E2 3312.981} C_VEL
LIN {X 0,Y 99.09,Z 948.377,A -85,B 0,C 180,E1 3311.189,E2 3311.189} C_VEL
LIN {X 0,Y 93.195,Z 962.718,A -85,B 0,C 180,E1 3308.934,E2 3308.934} C_VEL
LIN {X 0,Y 89.515,Z 970.625,A -85,B 0,C 180,E1 3307.112,E2 3307.112} C_VEL
LIN {X 0,Y 82.709,Z 986.213,A -85,B 0,C 180,E1 3305.014,E2 3305.014} C_VEL
LIN {X 0,Y 76.992,Z 997.463,A -85,B 0,C 180,E1 3301.983,E2 3301.983} C_VEL
LIN {X 0,Y 74.03,Z 1002.653,A -85,B 0,C 180,E1 3299.781,E2 3299.781} C_VEL
LIN {X 0,Y 68.558,Z 1013.339,A -85,B 0,C 180,E1 3296.958,E2 3296.958} C_VEL
LIN {X 0,Y 63.933,Z 1021.745,A -85,B 0,C 180,E1 3292.87,E2 3292.87} C_VEL
LIN {X 0,Y 62.372,Z 1024.453,A -85,B 0,C 180,E1 3290.999,E2 3290.999} C_VEL
LIN {X 0,Y 57.031,Z 1034.57,A -85,B 0,C 180,E1 3286.652,E2 3286.652} C_VEL
LIN {X 0,Y 53.318,Z 1041.67,A -85,B 0,C 180,E1 3280.991,E2 3280.991} C_VEL
LIN {X 0,Y 52.164,Z 1044.191,A -85,B 0,C 180,E1 3278.502,E2 3278.502} C_VEL
LIN {X 0,Y 47.764,Z 1053.464,A -85,B 0,C 180,E1 3271.526,E2 3271.526} C_VEL
LIN {X 0,Y 45.61,Z 1060.207,A -85,B 0,C 180,E1 3263.01,E2 3263.01} C_VEL
LIN {X 0,Y 45.252,Z 1062.907,A -85,B 0,C 180,E1 3258.657,E2 3258.657} C_VEL
LIN {X 0,Y 43.234,Z 1071.957,A -85,B 0,C 180,E1 3247.947,E2 3247.947} C_VEL
LIN {X 0,Y 44.031,Z 1078.843,A -85,B 0,C 180,E1 3237.252,E2 3237.252} C_VEL
LIN {X 0,Y 45.898,Z 1082.111,A -85,B 0,C 180,E1 3231.201,E2 3231.201} C_VEL
LIN {X 0,Y 49.006,Z 1093.063,A -85,B 0,C 180,E1 3217.164,E2 3217.164} C_VEL
LIN {X 0,Y 56.713,Z 1103.658,A -85,B 0,C 180,E1 3204.395,E2 3204.395} C_VEL
LIN {X 0,Y 62.564,Z 1108.778,A -85,B 0,C 180,E1 3198.996,E2 3198.996} C_VEL
LIN {X 0,Y 53.614,Z 1115.474,A -85,B 0,C 180,E1 3193.612,E2 3193.612} C_VEL
LIN {X 0,Y 44.869,Z 1124.54,A -85,B 0,C 180,E1 3182.311,E2 3182.311} C_VEL
LIN {X 0,Y 39.967,Z 1134.403,A -85,B 0,C 180,E1 3164.468,E2 3164.468} C_VEL
LIN {X 0,Y 42.456,Z 1147.081,A -85,B 0,C 180,E1 3137.744,E2 3137.744} C_VEL
LIN {X 0,Y 43.368,Z 1148.76,A -85,B 0,C 180,E1 3133.92,E2 3133.92} C_VEL
LIN {X 0,Y 48.491,Z 1155.619,A -85,B 0,C 180,E1 3108.692,E2 3108.692} C_VEL
LIN {X 0,Y 49.724,Z 1156.419,A -85,B 0,C 180,E1 3105.666,E2 3105.666} C_VEL
LIN {X 0,Y 41.281,Z 1147.912,A -85,B 0,C 180,E1 3085.881,E2 3085.881} C_VEL
LIN {X 0,Y 38.271,Z 1142.129,A -85,B 0,C 180,E1 3072.097,E2 3072.097} C_VEL
LIN {X 0,Y 36.715,Z 1131.363,A -85,B 0,C 180,E1 3048.749,E2 3048.749} C_VEL
LIN {X 0,Y 40.571,Z 1118.197,A -85,B 0,C 180,E1 3025.507,E2 3025.507} C_VEL
LIN {X 0,Y 49.783,Z 1101.862,A -85,B 0,C 180,E1 3007.071,E2 3007.071} C_VEL
LIN {X 0,Y 61.777,Z 1083.322,A -85,B 0,C 180,E1 2995.041,E2 2995.041} C_VEL
LIN {X 0,Y 74.371,Z 1063.243,A -85,B 0,C 180,E1 2987.398,E2 2987.398} C_VEL
LIN {X 0,Y 86.46,Z 1042.162,A -85,B 0,C 180,E1 2982.327,E2 2982.327} C_VEL
LIN {X 0,Y 98.087,Z 1019.054,A -85,B 0,C 180,E1 2978.671,E2 2978.671} C_VEL
LIN {X 0,Y 108.57,Z 994.887,A -85,B 0,C 180,E1 2976.056,E2 2976.056} C_VEL
LIN {X 0,Y 117.77,Z 969.441,A -85,B 0,C 180,E1 2974.137,E2 2974.137} C_VEL
LIN {X 0,Y 124.285,Z 947.393,A -85,B 0,C 180,E1 2972.953,E2 2972.953} C_VEL
LIN {X 0,Y 125.693,Z 939.919,A -85,B 0,C 180,E1 2972.259,E2 2972.259} C_VEL
LIN {X 0,Y 127.092,Z 919.849,A -85,B 0,C 180,E1 2969.134,E2 2969.134} C_VEL
LIN {X 0,Y 128.301,Z 913.399,A -85,B 0,C 180,E1 2968.599,E2 2968.599} C_VEL
LIN {X 0,Y 142.722,Z 857.175,A -85,B 0,C 180,E1 2966.592,E2 2966.592} C_VEL
LIN {X 0,Y 142.285,Z 856.234,A -85,B 0,C 180,E1 2966.125,E2 2966.125} C_VEL
LIN {X 0,Y 132.47,Z 874.726,A -85,B 0,C 180,E1 2963.144,E2 2963.144} C_VEL
LIN {X 0,Y 130.452,Z 878.763,A -85,B 0,C 180,E1 2962.53,E2 2962.53} C_VEL
LIN {X 0,Y 119.395,Z 904.372,A -85,B 0,C 180,E1 2959.679,E2 2959.679} C_VEL
LIN {X 0,Y 112.544,Z 921.768,A -85,B 0,C 180,E1 2958.011,E2 2958.011} C_VEL
LIN {X 0,Y 108.83,Z 930.413,A -85,B 0,C 180,E1 2956.823,E2 2956.823} C_VEL
LIN {X 0,Y 101.344,Z 951.084,A -85,B 0,C 180,E1 2955.303,E2 2955.303} C_VEL
LIN {X 0,Y 94.966,Z 965.754,A -85,B 0,C 180,E1 2953.312,E2 2953.312} C_VEL
LIN {X 0,Y 91.039,Z 973.795,A -85,B 0,C 180,E1 2951.765,E2 2951.765} C_VEL
LIN {X 0,Y 84,Z 989.117,A -85,B 0,C 180,E1 2950.067,E2 2950.067} C_VEL
LIN {X 0,Y 77.889,Z 1000.302,A -85,B 0,C 180,E1 2947.517,E2 2947.517} C_VEL
LIN {X 0,Y 74.211,Z 1006.492,A -85,B 0,C 180,E1 2945.389,E2 2945.389} C_VEL
LIN {X 0,Y 68.011,Z 1017.532,A -85,B 0,C 180,E1 2942.764,E2 2942.764} C_VEL
LIN {X 0,Y 62.556,Z 1026.286,A -85,B 0,C 180,E1 2938.735,E2 2938.735} C_VEL
LIN {X 0,Y 61.023,Z 1028.792,A -85,B 0,C 180,E1 2937.509,E2 2937.509} C_VEL
LIN {X 0,Y 55.246,Z 1038.442,A -85,B 0,C 180,E1 2933.61,E2 2933.61} C_VEL
LIN {X 0,Y 50.808,Z 1045.797,A -85,B 0,C 180,E1 2928.023,E2 2928.023} C_VEL
LIN {X 0,Y 49.36,Z 1048.225,A -85,B 0,C 180,E1 2925.944,E2 2925.944} C_VEL
LIN {X 0,Y 43.994,Z 1057.759,A -85,B 0,C 180,E1 2918.646,E2 2918.646} C_VEL
LIN {X 0,Y 40.916,Z 1064.688,A -85,B 0,C 180,E1 2909.223,E2 2909.223} C_VEL
LIN {X 0,Y 40.354,Z 1066.703,A -85,B 0,C 180,E1 2905.662,E2 2905.662} C_VEL
LIN {X 0,Y 37.26,Z 1076.485,A -85,B 0,C 180,E1 2892.363,E2 2892.363} C_VEL
LIN {X 0,Y 37.54,Z 1083.11,A -85,B 0,C 180,E1 2879.967,E2 2879.967} C_VEL
LIN {X 0,Y 39.07,Z 1086.61,A -85,B 0,C 180,E1 2872.616,E2 2872.616} C_VEL
LIN {X 0,Y 41.751,Z 1096.438,A -85,B 0,C 180,E1 2857.437,E2 2857.437} C_VEL
LIN {X 0,Y 49.512,Z 1107.006,A -85,B 0,C 180,E1 2842.679,E2 2842.679} C_VEL
LIN {X 0,Y 51.336,Z 1108.852,A -85,B 0,C 180,E1 2840.487,E2 2840.487} C_VEL
LIN {X 0,Y 41.175,Z 1117.633,A -85,B 0,C 180,E1 2830.945,E2 2830.945} C_VEL
LIN {X 0,Y 33.452,Z 1128.378,A -85,B 0,C 180,E1 2810.994,E2 2810.994} C_VEL
LIN {X 0,Y 34.519,Z 1141.549,A -85,B 0,C 180,E1 2778.278,E2 2778.278} C_VEL
LIN {X 0,Y 36.828,Z 1145.245,A -85,B 0,C 180,E1 2769.31,E2 2769.31} C_VEL
LIN {X 0,Y 41.44,Z 1150.661,A -85,B 0,C 180,E1 2746.969,E2 2746.969} C_VEL
LIN {X 0,Y 33.619,Z 1142.704,A -85,B 0,C 180,E1 2726.536,E2 2726.536} C_VEL
LIN {X 0,Y 29.791,Z 1134.813,A -85,B 0,C 180,E1 2705.821,E2 2705.821} C_VEL
LIN {X 0,Y 30.443,Z 1122.241,A -85,B 0,C 180,E1 2674.769,E2 2674.769} C_VEL
LIN {X 0,Y 37.985,Z 1107.586,A -85,B 0,C 180,E1 2650.29,E2 2650.29} C_VEL
LIN {X 0,Y 49.712,Z 1090.295,A -85,B 0,C 180,E1 2635.002,E2 2635.002} C_VEL
LIN {X 0,Y 62.866,Z 1070.916,A -85,B 0,C 180,E1 2625.867,E2 2625.867} C_VEL
LIN {X 0,Y 75.666,Z 1050.391,A -85,B 0,C 180,E1 2620.208,E2 2620.208} C_VEL
LIN {X 0,Y 87.521,Z 1028.953,A -85,B 0,C 180,E1 2616.45,E2 2616.45} C_VEL
LIN {X 0,Y 98.674,Z 1005.689,A -85,B 0,C 180,E1 2613.724,E2 2613.724} C_VEL
LIN {X 0,Y 108.763,Z 980.653,A -85,B 0,C 180,E1 2611.724,E2 2611.724} C_VEL
LIN {X 0,Y 117.214,Z 955.05,A -85,B 0,C 180,E1 2610.282,E2 2610.282} C_VEL
LIN {X 0,Y 128.301,Z 913.399,A -85,B 0,C 180,E1 2608.599,E2 2608.599} C_VEL
LIN {X 0,Y 129.044,Z 908.369,A -85,B 0,C 180,E1 2608.037,E2 2608.037} C_VEL
LIN {X 0,Y 129.07,Z 895.318,A -85,B 0,C 180,E1 2605.265,E2 2605.265} C_VEL
LIN {X 0,Y 129.795,Z 890.995,A -85,B 0,C 180,E1 2604.835,E2 2604.835} C_VEL
LIN {X 0,Y 130.176,Z 889.373,A -85,B 0,C 180,E1 2604.75,E2 2604.75} C_VEL
LIN {X 0,Y 122.388,Z 907.189,A -85,B 0,C 180,E1 2602.95,E2 2602.95} C_VEL
LIN {X 0,Y 115.238,Z 924.856,A -85,B 0,C 180,E1 2601.47,E2 2601.47} C_VEL
LIN {X 0,Y 111.685,Z 933.06,A -85,B 0,C 180,E1 2600.493,E2 2600.493} C_VEL
LIN {X 0,Y 104.219,Z 953.255,A -85,B 0,C 180,E1 2599.288,E2 2599.288} C_VEL
LIN {X 0,Y 97.259,Z 968.694,A -85,B 0,C 180,E1 2597.533,E2 2597.533} C_VEL
LIN {X 0,Y 93.621,Z 975.645,A -85,B 0,C 180,E1 2596.322,E2 2596.322} C_VEL
LIN {X 0,Y 86.375,Z 990.929,A -85,B 0,C 180,E1 2595.091,E2 2595.091} C_VEL
LIN {X 0,Y 79.929,Z 1002.344,A -85,B 0,C 180,E1 2593.079,E2 2593.079} C_VEL
LIN {X 0,Y 75.074,Z 1010.057,A -85,B 0,C 180,E1 2590.965,E2 2590.965} C_VEL
LIN {X 0,Y 68.155,Z 1021.605,A -85,B 0,C 180,E1 2588.631,E2 2588.631} C_VEL
LIN {X 0,Y 60.946,Z 1032.161,A -85,B 0,C 180,E1 2584.418,E2 2584.418} C_VEL
LIN {X 0,Y 54.311,Z 1042.255,A -85,B 0,C 180,E1 2580.937,E2 2580.937} C_VEL
LIN {X 0,Y 48.63,Z 1050.231,A -85,B 0,C 180,E1 2575.284,E2 2575.284} C_VEL
LIN {X 0,Y 40.953,Z 1061.842,A -85,B 0,C 180,E1 2567.048,E2 2567.048} C_VEL
LIN {X 0,Y 36.685,Z 1069.146,A -85,B 0,C 180,E1 2556.801,E2 2556.801} C_VEL
LIN {X 0,Y 35.549,Z 1071.379,A -85,B 0,C 180,E1 2553.22,E2 2553.22} C_VEL
LIN {X 0,Y 31.532,Z 1080.852,A -85,B 0,C 180,E1 2538.446,E2 2538.446} C_VEL
LIN {X 0,Y 31.301,Z 1088.094,A -85,B 0,C 180,E1 2521.791,E2 2521.791} C_VEL
LIN {X 0,Y 32.243,Z 1090.991,A -85,B 0,C 180,E1 2514.623,E2 2514.623} C_VEL
LIN {X 0,Y 35.802,Z 1102.157,A -85,B 0,C 180,E1 2493.42,E2 2493.42} C_VEL
LIN {X 0,Y 40.813,Z 1108.892,A -85,B 0,C 180,E1 2482.396,E2 2482.396} C_VEL
LIN {X 0,Y 29.967,Z 1119.2,A -85,B 0,C 180,E1 2466.879,E2 2466.879} C_VEL
LIN {X 0,Y 25.096,Z 1130.679,A -85,B 0,C 180,E1 2434.513,E2 2434.513} C_VEL
LIN {X 0,Y 30.699,Z 1141.57,A -85,B 0,C 180,E1 2402.843,E2 2402.843} C_VEL
LIN {X 0,Y 33.241,Z 1144.428,A -85,B 0,C 180,E1 2388.818,E2 2388.818} C_VEL
LIN {X 0,Y 26.823,Z 1138.174,A -85,B 0,C 180,E1 2371.512,E2 2371.512} C_VEL
LIN {X 0,Y 22.18,Z 1129.787,A -85,B 0,C 180,E1 2345.229,E2 2345.229} C_VEL
LIN {X 0,Y 24.199,Z 1116.664,A -85,B 0,C 180,E1 2304.721,E2 2304.721} C_VEL
LIN {X 0,Y 34.692,Z 1100.594,A -85,B 0,C 180,E1 2278.547,E2 2278.547} C_VEL
LIN {X 0,Y 47.94,Z 1082.78,A -85,B 0,C 180,E1 2265.749,E2 2265.749} C_VEL
LIN {X 0,Y 61.192,Z 1063.872,A -85,B 0,C 180,E1 2258.807,E2 2258.807} C_VEL
LIN {X 0,Y 74.675,Z 1042.254,A -85,B 0,C 180,E1 2254.261,E2 2254.261} C_VEL
LIN {X 0,Y 86.717,Z 1019.989,A -85,B 0,C 180,E1 2251.33,E2 2251.33} C_VEL
LIN {X 0,Y 97.975,Z 995.532,A -85,B 0,C 180,E1 2249.207,E2 2249.207} C_VEL
LIN {X 0,Y 107.824,Z 969.782,A -85,B 0,C 180,E1 2247.669,E2 2247.669} C_VEL
LIN {X 0,Y 115.982,Z 942.977,A -85,B 0,C 180,E1 2246.579,E2 2246.579} C_VEL
LIN {X 0,Y 129.795,Z 890.995,A -85,B 0,C 180,E1 2244.835,E2 2244.835} C_VEL
LIN {X 0,Y 133.586,Z 891.523,A -85,B 0,C 180,E1 2244.386,E2 2244.386} C_VEL
LIN {X 0,Y 133.586,Z 977.645,A -85,B 0,C 180,E1 2244.386,E2 2244.386} C_VEL
LIN {X 0,Y 114.863,Z 977.645,A -85,B 0,C 180,E1 2244.279,E2 2244.279} C_VEL
LIN {X 0,Y 112.863,Z 975.645,A -85,B 0,C 180,E1 2244.265,E2 2244.265} C_VEL
LIN {X 0,Y 112.863,Z 951.35,A -85,B 0,C 180,E1 2244.265,E2 2244.265} C_VEL
LIN {X 0,Y 109.515,Z 950.392,A -85,B 0,C 180,E1 2243.388,E2 2243.388} C_VEL
LIN {X 0,Y 101.95,Z 967.662,A -85,B 0,C 180,E1 2242.03,E2 2242.03} C_VEL
LIN {X 0,Y 95.757,Z 979.494,A -85,B 0,C 180,E1 2240.579,E2 2240.579} C_VEL
LIN {X 0,Y 87.919,Z 995.398,A -85,B 0,C 180,E1 2239.571,E2 2239.571} C_VEL
LIN {X 0,Y 80.337,Z 1007.816,A -85,B 0,C 180,E1 2237.617,E2 2237.617} C_VEL
LIN {X 0,Y 77.101,Z 1012.526,A -85,B 0,C 180,E1 2236.493,E2 2236.493} C_VEL
LIN {X 0,Y 69.907,Z 1024.057,A -85,B 0,C 180,E1 2234.824,E2 2234.824} C_VEL
LIN {X 0,Y 61.726,Z 1035.298,A -85,B 0,C 180,E1 2231.31,E2 2231.31} C_VEL
LIN {X 0,Y 54.708,Z 1045.324,A -85,B 0,C 180,E1 2228.701,E2 2228.701} C_VEL
LIN {X 0,Y 47.906,Z 1053.854,A -85,B 0,C 180,E1 2223.769,E2 2223.769} C_VEL
LIN {X 0,Y 39.279,Z 1065.3,A -85,B 0,C 180,E1 2217.085,E2 2217.085} C_VEL
LIN {X 0,Y 33.172,Z 1073.436,A -85,B 0,C 180,E1 2206.283,E2 2206.283} C_VEL
LIN {X 0,Y 26.225,Z 1085.015,A -85,B 0,C 180,E1 2187.174,E2 2187.174} C_VEL
LIN {X 0,Y 24.859,Z 1092.157,A -85,B 0,C 180,E1 2166.88,E2 2166.88} C_VEL
LIN {X 0,Y 25.366,Z 1095.107,A -85,B 0,C 180,E1 2157.692,E2 2157.692} C_VEL
LIN {X 0,Y 28.407,Z 1105.248,A -85,B 0,C 180,E1 2132.72,E2 2132.72} C_VEL
LIN {X 0,Y 30.719,Z 1108.875,A -85,B 0,C 180,E1 2125.227,E2 2125.227} C_VEL
LIN {X 0,Y 19.886,Z 1119.987,A -85,B 0,C 180,E1 2100.14,E2 2100.14} C_VEL
LIN {X 0,Y 19.757,Z 1131.541,A -85,B 0,C 180,E1 2052.281,E2 2052.281} C_VEL
LIN {X 0,Y 25.265,Z 1137.837,A -85,B 0,C 180,E1 2032.406,E2 2032.406} C_VEL
LIN {X 0,Y 19.007,Z 1132.033,A -85,B 0,C 180,E1 2015.435,E2 2015.435} C_VEL
LIN {X 0,Y 14.294,Z 1121.239,A -85,B 0,C 180,E1 1967.975,E2 1967.975} C_VEL
LIN {X 0,Y 22.843,Z 1105.779,A -85,B 0,C 180,E1 1919.015,E2 1919.015} C_VEL
LIN {X 0,Y 36.399,Z 1089.1,A -85,B 0,C 180,E1 1902.347,E2 1902.347} C_VEL
LIN {X 0,Y 50.159,Z 1071.146,A -85,B 0,C 180,E1 1894.952,E2 1894.952} C_VEL
LIN {X 0,Y 64.971,Z 1049.337,A -85,B 0,C 180,E1 1890.339,E2 1890.339} C_VEL
LIN {X 0,Y 77.531,Z 1027.928,A -85,B 0,C 180,E1 1887.691,E2 1887.691} C_VEL
LIN {X 0,Y 89.204,Z 1004.69,A -85,B 0,C 180,E1 1885.819,E2 1885.819} C_VEL
LIN {X 0,Y 99.168,Z 981.109,A -85,B 0,C 180,E1 1884.52,E2 1884.52} C_VEL
LIN {X 0,Y 107.962,Z 955.634,A -85,B 0,C 180,E1 1883.542,E2 1883.542} C_VEL
LIN {X 0,Y 109.515,Z 950.392,A -85,B 0,C 180,E1 1883.388,E2 1883.388} C_VEL
LIN {X 0,Y 113.373,Z 950.973,A -85,B 0,C 180,E1 1883.046,E2 1883.046} C_VEL
LIN {X 0,Y 113.373,Z 1033.245,A -85,B 0,C 180,E1 1883.046,E2 1883.046} C_VEL
LIN {X 0,Y 85.178,Z 1033.245,A -85,B 0,C 180,E1 1882.814,E2 1882.814} C_VEL
LIN {X 0,Y 83.178,Z 1031.245,A -85,B 0,C 180,E1 1882.791,E2 1882.791} C_VEL
LIN {X 0,Y 83.178,Z 1016.004,A -85,B 0,C 180,E1 1882.791,E2 1882.791} C_VEL
LIN {X 0,Y 79.951,Z 1014.718,A -85,B 0,C 180,E1 1881.783,E2 1881.783} C_VEL
LIN {X 0,Y 71.453,Z 1027.735,A -85,B 0,C 180,E1 1880.481,E2 1880.481} C_VEL
LIN {X 0,Y 63.359,Z 1038.277,A -85,B 0,C 180,E1 1877.983,E2 1877.983} C_VEL
LIN {X 0,Y 55.583,Z 1048.752,A -85,B 0,C 180,E1 1876.168,E2 1876.168} C_VEL
LIN {X 0,Y 47.275,Z 1058.48,A -85,B 0,C 180,E1 1872.046,E2 1872.046} C_VEL
LIN {X 0,Y 38.867,Z 1068.63,A -85,B 0,C 180,E1 1867.751,E2 1867.751} C_VEL
LIN {X 0,Y 31.447,Z 1076.808,A -85,B 0,C 180,E1 1859.068,E2 1859.068} C_VEL
LIN {X 0,Y 29.053,Z 1079.638,A -85,B 0,C 180,E1 1855.611,E2 1855.611} C_VEL
LIN {X 0,Y 21.791,Z 1089.107,A -85,B 0,C 180,E1 1839.894,E2 1839.894} C_VEL
LIN {X 0,Y 18.649,Z 1096.819,A -85,B 0,C 180,E1 1812.316,E2 1812.316} C_VEL
LIN {X 0,Y 18.603,Z 1099.165,A -85,B 0,C 180,E1 1803.014,E2 1803.014} C_VEL
LIN {X 0,Y 21.086,Z 1108.701,A -85,B 0,C 180,E1 1770.45,E2 1770.45} C_VEL
LIN {X 0,Y 10.848,Z 1120.737,A -85,B 0,C 180,E1 1720.549,E2 1720.549} C_VEL
LIN {X 0,Y 14.294,Z 1128.12,A -85,B 0,C 180,E1 1674.894,E2 1674.894} C_VEL
LIN {X 0,Y 7.158,Z 1116.314,A -85,B 0,C 180,E1 1595.414,E2 1595.414} C_VEL
LIN {X 0,Y 18.631,Z 1101.909,A -85,B 0,C 180,E1 1541.958,E2 1541.958} C_VEL
LIN {X 0,Y 34.476,Z 1083.996,A -85,B 0,C 180,E1 1530.64,E2 1530.64} C_VEL
LIN {X 0,Y 49.579,Z 1064.614,A -85,B 0,C 180,E1 1526.23,E2 1526.23} C_VEL
LIN {X 0,Y 63.341,Z 1044.23,A -85,B 0,C 180,E1 1523.799,E2 1523.799} C_VEL
LIN {X 0,Y 76.176,Z 1022.019,A -85,B 0,C 180,E1 1522.185,E2 1522.185} C_VEL
LIN {X 0,Y 79.951,Z 1014.718,A -85,B 0,C 180,E1 1521.783,E2 1521.783} C_VEL
LIN {X 0,Y 83.697,Z 1015.627,A -85,B 0,C 180,E1 1521.421,E2 1521.421} C_VEL
LIN {X 0,Y 83.697,Z 1086.702,A -85,B 0,C 180,E1 1521.421,E2 1521.421} C_VEL
LIN {X 0,Y 44.048,Z 1086.702,A -85,B 0,C 180,E1 1519.617,E2 1519.617} C_VEL
LIN {X 0,Y 42.053,Z 1084.702,A -85,B 0,C 180,E1 1519.436,E2 1519.436} C_VEL
LIN {X 0,Y 42.053,Z 1074.202,A -85,B 0,C 180,E1 1519.436,E2 1519.436} C_VEL
LIN {X 0,Y 38.824,Z 1072.762,A -85,B 0,C 180,E1 1517.98,E2 1517.98} C_VEL
LIN {X 0,Y 29.129,Z 1082.211,A -85,B 0,C 180,E1 1510.599,E2 1510.599} C_VEL
LIN {X 0,Y 19.643,Z 1092.084,A -85,B 0,C 180,E1 1499.793,E2 1499.793} C_VEL
LIN {X 0,Y 13.242,Z 1099.937,A -85,B 0,C 180,E1 1471.798,E2 1471.798} C_VEL
LIN {X 0,Y 12.403,Z 1102.055,A -85,B 0,C 180,E1 1458.707,E2 1458.707} C_VEL
LIN {X 0,Y 11.973,Z 1108.504,A -85,B 0,C 180,E1 1423.085,E2 1423.085} C_VEL
LIN {X 0,Y 3.607,Z 1116.9,A -85,B 0,C 180,E1 1349.407,E2 1349.407} C_VEL
LIN {X 0,Y 12.227,Z 1102.477,A -85,B 0,C 180,E1 1518.378,E2 1518.378} C_VEL
LIN {X 0,Y 28.558,Z 1085.156,A -85,B 0,C 180,E1 1518.401,E2 1518.401} C_VEL
LIN {X 0,Y 38.824,Z 1072.762,A -85,B 0,C 180,E1 1517.98,E2 1517.98} C_VEL
LIN {X 0,Y 39.665,Z 1074.215,A -85,B 0,C 180,E1 1513.207,E2 1513.207} C_VEL
LIN {X 0,Y 39.665,Z 1240.5,A -85,B 0,C 180,E1 1513.207,E2 1513.207} C_VEL
LIN {X 0,Y 39.665,Z 1240.5,A -85,B 0,C 180,E1 1513.207,E2 1513.207}

QRS_NEXT_CUT()

QRS_NEXT()
QRS_HOME()

END
